(* CODESYS project ugp_spk.project

Project tree, tasks and I/O mapping:
  Device : Owen SPK2xx 03.CS.WEB, Owen, order no. 023, version 3.5.4.20
    application Application
      libraries: Standard, * (System); Util, 3.5.1.0 (System); CmpSysExec, 1.0.0.2 (Owen); ArchiverSPK, 3.5.3.53 (Owen); VisuDialogs, * (System)
      task MainTask (cyclic, interval t#100ms, priority 2) calls PLC_PRG, InterviewState
      task VISU_TASK (cyclic, interval 100 ms, priority 30) calls VisuElems.Visu_Prg
      task AlarmManagerTask (cyclic, interval 50 ms, priority 31) calls AlarmManager.Alarm_Prg
      task bus_task (cyclic, interval t#100ms, priority 1, watchdog t#1000ms x 1) calls MV110
      task LogTask (cyclic, interval t#10000ms, priority 5) calls LogSaver
      program PLC_PRG [ST]
      Alarm Configuration
        alarm class Error (priority 10, acknowledge REP_ACK)
        alarm class Warning (priority 30, acknowledge REP)
        AlarmStorage
        text list AlarmGroup
        alarm group AlarmGroup
            19 [Warning]: Comparison Equal, ExpressionToCompare TRUE, Expression InterviewState.MV110_err - "Нет связи с ЩРПА, ШАСН, ШОПС"
            10 [Warning]: Comparison Equal, ExpressionToCompare TRUE, Expression PLC_PRG.mv110_in_0_alarm_shos - "Нарушение ШОС"
            11 [Warning]: Comparison Equal, ExpressionToCompare TRUE, Expression PLC_PRG.mv110_in_2_alarm_ops - "Авария ОПС"
            12 [Warning]: Comparison Equal, ExpressionToCompare TRUE, Expression PLC_PRG.mpx1_alarm - "Авария ИБПC 2.1"
            13 [Warning]: Comparison Equal, ExpressionToCompare TRUE, Expression PLC_PRG.mpx2_alarm - "Авария ИБПC 2.2"
            14 [Warning]: Comparison Equal, ExpressionToCompare TRUE, Expression PLC_PRG.mv110_in_7_heating - "Обогрев"
            15 [Warning]: Comparison Equal, ExpressionToCompare TRUE, Expression InterviewState.IPS1_err - "Нет связи с ИБПА 1.1"
            16 [Warning]: Comparison Equal, ExpressionToCompare TRUE, Expression InterviewState.IPS2_err - "Нет связи с ИБПА 1.2"
            17 [Warning]: Comparison Equal, ExpressionToCompare TRUE, Expression InterviewState.MPX1_err - "Нет связи с ИБПС 2.1"
            18 [Warning]: Comparison Equal, ExpressionToCompare TRUE, Expression InterviewState.MPX2_err - "Нет связи с ИБПС 2.2"
            9 [Warning]: Comparison Equal, ExpressionToCompare TRUE, Expression PLC_PRG.mv110_in_1_fire - "Пожар"
            20 [Warning]: Comparison Equal, ExpressionToCompare TRUE, Expression PLC_PRG.climate_temp_excess - "Превышена максимальная температура"
      function block Two_words_to_Real [ST]
      visualisation mpx_1_params
      visualisation SCHRPA
      image pool ImagePool
      visualisation mpx_1_state
      visualisation mpx_2_params
      visualisation mpx_2_state
      visualisation main
      visualisation climate
      visualisation SHASN
      visualisation ips_1
      visualisation ips_2
      visualisation alarms
      visualisation log_data
      visualisation SHOPS
      program InterviewState [ST]
      program LogSaver [ST]
    Modbus_COM : Modbus COM, 3S - Smart Software Solutions GmbH, version 3.4.0.0
        settings: DataBits = 8; StopBits = 1; ComPort = 3
      Modbus_Master_COM_Port : Modbus Master, COM Port, 3S - Smart Software Solutions GmbH, version 3.5.5.0
          settings: Transmission = 'RTU'; ResponseTimeout = 1000; TimeBetweenFrames = 10; Auto-restart communication = TRUE
        MV110 : Modbus Slave, COM Port, 3S - Smart Software Solutions GmbH, version 3.5.4.0
            settings: SlaveAddress = 10; ResponseTimeout = 1000; UseExtendedFunctionCodes = TRUE; Channel 0.Function Code = 3; Channel 0.Read Offset = 16#0033; Channel 0.Read Length = 1; Channel 0.Write Offset = 0; Channel 0.Write Length = 0; Channel 0.Cycle Time = 100
            input  Application.PLC_PRG.mv110_reg : WORD  // Channel 0.Channel 0
            unmapped channels: Channel 0
        MPX_1 : Modbus Slave, COM Port, 3S - Smart Software Solutions GmbH, version 3.5.4.0
            settings: SlaveAddress = 11; ResponseTimeout = 1000; UseExtendedFunctionCodes = TRUE; Input_group.Function Code = 4; Input_group.Read Offset = 16#000B; Input_group.Read Length = 7; Input_group.Write Offset = 0; Input_group.Write Length = 0; Input_group.Cycle Time = 300; Bypass_out_group.Function Code = 3; Bypass_out_group.Read Offset = 16#0015; Bypass_out_group.Read Length = 7; Bypass_out_group.Write Offset = 0; Bypass_out_group.Write Length = 0; Bypass_out_group.Cycle Time = 300; Output_group.Function Code = 3; Output_group.Read Offset = 16#001F; Output_group.Read Length = 13; Output_group.Write Offset = 0; Output_group.Write Length = 0; Output_group.Cycle Time = 300; Battery_group.Function Code = 3; Battery_group.Read Offset = 16#002F; Battery_group.Read Length = 7; Battery_group.Write Offset = 0; Battery_group.Write Length = 0; Battery_group.Cycle Time = 300; temp.Function Code = 3; temp.Read Offset = 16#003D; temp.Read Length = 1; temp.Write Offset = 0; temp.Write Length = 0; temp.Cycle Time = 300; states.Function Code = 3; states.Read Offset = 16#0000; states.Read Length = 2; states.Write Offset = 0; states.Write Length = 0; states.Cycle Time = 300; Channel 6.Function Code = 6;
              Channel 6.Read Offset = 0; Channel 6.Read Length = 0; Channel 6.Write Offset = 16#0070; Channel 6.Write Length = 1; Channel 6.Cycle Time = 100
            input  Application.PLC_PRG.mpx1_in_v_1 : WORD  // Input_group.Input_group
            input  Application.PLC_PRG.mpx1_in_v_2 : WORD  // Input_group.Input_group
            input  Application.PLC_PRG.mpx1_in_v_3 : WORD  // Input_group.Input_group
            input  Application.PLC_PRG.mpx1_in_freq : WORD  // Input_group.Input_group
            input  Application.PLC_PRG.mpx1_bypass_v_1 : WORD  // Bypass_out_group.Bypass_out_group
            input  Application.PLC_PRG.mpx1_bypass_v_2 : WORD  // Bypass_out_group.Bypass_out_group
            input  Application.PLC_PRG.mpx1_bypass_v_3 : WORD  // Bypass_out_group.Bypass_out_group
            input  Application.PLC_PRG.mpx1_bypass_freq : WORD  // Bypass_out_group.Bypass_out_group
            input  Application.PLC_PRG.mpx1_output_v_1 : WORD  // Bypass_out_group.Bypass_out_group
            input  Application.PLC_PRG.mpx1_output_v_2 : WORD  // Bypass_out_group.Bypass_out_group
            input  Application.PLC_PRG.mpx1_output_v_3 : WORD  // Bypass_out_group.Bypass_out_group
            input  Application.PLC_PRG.mpx1_output_i_1 : WORD  // Output_group.Output_group
            input  Application.PLC_PRG.mpx1_output_i_2 : WORD  // Output_group.Output_group
            input  Application.PLC_PRG.mpx1_output_i_3 : WORD  // Output_group.Output_group
            input  Application.PLC_PRG.mpx1_load_ph_1 : WORD  // Output_group.Output_group
            input  Application.PLC_PRG.mpx1_load_ph_2 : WORD  // Output_group.Output_group
            input  Application.PLC_PRG.mpx1_load_ph_3 : WORD  // Output_group.Output_group
            input  Application.PLC_PRG.mpx1_output_active_power_1 : WORD  // Output_group.Output_group
            input  Application.PLC_PRG.mpx1_output_active_power_2 : WORD  // Output_group.Output_group
            input  Application.PLC_PRG.mpx1_output_active_power_3 : WORD  // Output_group.Output_group
            input  Application.PLC_PRG.mpx1_output_freq : WORD  // Output_group.Output_group
            input  Application.PLC_PRG.mpx1_battery_voltage : WORD  // Battery_group.Battery_group
            input  Application.PLC_PRG.mpx1_battery_current : WORD  // Battery_group.Battery_group
            input  Application.PLC_PRG.mpx1_battery_capacity : WORD  // Battery_group.Battery_group
            input  Application.PLC_PRG.mpx1_battery_time : WORD  // Battery_group.Battery_group
            input  Application.PLC_PRG.mpx1_temp : WORD  // temp.temp
            input  Application.PLC_PRG.mpx1_state_reg_1 : WORD  // states.states
            input  Application.PLC_PRG.mpx1_state_reg_2 : WORD  // states.states
            output Application.PLC_PRG.mpx_test_battery_start : BIT  // Channel 6
            output Application.PLC_PRG.mpx_test_battery_command : ARRAY[0..0] OF WORD  // Channel 6
            unmapped channels: Input_group, Bypass_out_group, Output_group, Battery_group, temp, states
        MPX_2 : Modbus Slave, COM Port, 3S - Smart Software Solutions GmbH, version 3.5.4.0
            settings: SlaveAddress = 12; ResponseTimeout = 1000; UseExtendedFunctionCodes = TRUE; Input_group.Function Code = 4; Input_group.Read Offset = 16#000B; Input_group.Read Length = 7; Input_group.Write Offset = 0; Input_group.Write Length = 0; Input_group.Cycle Time = 300; Bypass_out_group.Function Code = 3; Bypass_out_group.Read Offset = 16#0015; Bypass_out_group.Read Length = 7; Bypass_out_group.Write Offset = 0; Bypass_out_group.Write Length = 0; Bypass_out_group.Cycle Time = 300; Output_group.Function Code = 3; Output_group.Read Offset = 16#001F; Output_group.Read Length = 13; Output_group.Write Offset = 0; Output_group.Write Length = 0; Output_group.Cycle Time = 300; Battery_group.Function Code = 3; Battery_group.Read Offset = 16#002F; Battery_group.Read Length = 7; Battery_group.Write Offset = 0; Battery_group.Write Length = 0; Battery_group.Cycle Time = 300; temp.Function Code = 3; temp.Read Offset = 16#003D; temp.Read Length = 1; temp.Write Offset = 0; temp.Write Length = 0; temp.Cycle Time = 300; states.Function Code = 3; states.Read Offset = 16#0000; states.Read Length = 2; states.Write Offset = 0; states.Write Length = 0; states.Cycle Time = 300; Channel 6.Function Code = 6;
              Channel 6.Read Offset = 0; Channel 6.Read Length = 0; Channel 6.Write Offset = 16#0070; Channel 6.Write Length = 1; Channel 6.Cycle Time = 100
            input  Application.PLC_PRG.mpx2_in_v_1 : WORD  // Input_group.Input_group
            input  Application.PLC_PRG.mpx2_in_v_2 : WORD  // Input_group.Input_group
            input  Application.PLC_PRG.mpx2_in_v_3 : WORD  // Input_group.Input_group
            input  Application.PLC_PRG.mpx2_in_freq : WORD  // Input_group.Input_group
            input  Application.PLC_PRG.mpx2_bypass_v_1 : WORD  // Bypass_out_group.Bypass_out_group
            input  Application.PLC_PRG.mpx2_bypass_v_2 : WORD  // Bypass_out_group.Bypass_out_group
            input  Application.PLC_PRG.mpx2_bypass_v_3 : WORD  // Bypass_out_group.Bypass_out_group
            input  Application.PLC_PRG.mpx2_bypass_freq : WORD  // Bypass_out_group.Bypass_out_group
            input  Application.PLC_PRG.mpx2_output_v_1 : WORD  // Bypass_out_group.Bypass_out_group
            input  Application.PLC_PRG.mpx2_output_v_2 : WORD  // Bypass_out_group.Bypass_out_group
            input  Application.PLC_PRG.mpx2_output_v_3 : WORD  // Bypass_out_group.Bypass_out_group
            input  Application.PLC_PRG.mpx2_output_i_1 : WORD  // Output_group.Output_group
            input  Application.PLC_PRG.mpx2_output_i_2 : WORD  // Output_group.Output_group
            input  Application.PLC_PRG.mpx2_output_i_3 : WORD  // Output_group.Output_group
            input  Application.PLC_PRG.mpx2_load_ph_1 : WORD  // Output_group.Output_group
            input  Application.PLC_PRG.mpx2_load_ph_2 : WORD  // Output_group.Output_group
            input  Application.PLC_PRG.mpx2_load_ph_3 : WORD  // Output_group.Output_group
            input  Application.PLC_PRG.mpx2_output_active_power_1 : WORD  // Output_group.Output_group
            input  Application.PLC_PRG.mpx2_output_active_power_2 : WORD  // Output_group.Output_group
            input  Application.PLC_PRG.mpx2_output_active_power_3 : WORD  // Output_group.Output_group
            input  Application.PLC_PRG.mpx2_output_freq : WORD  // Output_group.Output_group
            input  Application.PLC_PRG.mpx2_battery_voltage : WORD  // Battery_group.Battery_group
            input  Application.PLC_PRG.mpx2_battery_current : WORD  // Battery_group.Battery_group
            input  Application.PLC_PRG.mpx2_battery_capacity : WORD  // Battery_group.Battery_group
            input  Application.PLC_PRG.mpx2_battery_time : WORD  // Battery_group.Battery_group
            input  Application.PLC_PRG.mpx2_temp : WORD  // temp.temp
            input  Application.PLC_PRG.mpx2_state_reg_1 : WORD  // states.states
            input  Application.PLC_PRG.mpx2_state_reg_2 : WORD  // states.states
            output Application.PLC_PRG.mpx_test_battery_start : BIT  // Channel 6
            output Application.PLC_PRG.mpx_test_battery_command : ARRAY[0..0] OF WORD  // Channel 6
            unmapped channels: Input_group, Bypass_out_group, Output_group, Battery_group, temp, states
    Modbus_slave : Modbus COM, 3S - Smart Software Solutions GmbH, version 3.4.0.0
        settings: DataBits = 8; StopBits = 1; ComPort = 4
      Modbus_Serial_Device : Modbus Serial Device, 3S - Smart Software Solutions GmbH, version 3.5.3.80
          settings: Unit-ID = 3
          output Application.PLC_PRG.mpx1_battery_capacity : WORD  // Outputs.Outputs
          output Application.PLC_PRG.mpx1_battery_current : WORD  // Outputs.Outputs
          output Application.PLC_PRG.mpx1_battery_time : WORD  // Outputs.Outputs
          output Application.PLC_PRG.mpx1_battery_voltage : WORD  // Outputs.Outputs
          output Application.PLC_PRG.mpx1_bypass_freq : WORD  // Outputs.Outputs
          output Application.PLC_PRG.mpx1_bypass_v_1 : WORD  // Outputs.Outputs
          output Application.PLC_PRG.mpx1_bypass_v_2 : WORD  // Outputs.Outputs
          output Application.PLC_PRG.mpx1_bypass_v_3 : WORD  // Outputs.Outputs
          output Application.PLC_PRG.mpx1_in_freq : WORD  // Outputs.Outputs
          output Application.PLC_PRG.mpx1_in_v_1 : WORD  // Outputs.Outputs
          output Application.PLC_PRG.mpx1_in_v_2 : WORD  // Outputs.Outputs
          output Application.PLC_PRG.mpx1_in_v_3 : WORD  // Outputs.Outputs
          output Application.PLC_PRG.mpx1_load_ph_1 : WORD  // Outputs.Outputs
          output Application.PLC_PRG.mpx1_load_ph_2 : WORD  // Outputs.Outputs
          output Application.PLC_PRG.mpx1_load_ph_3 : WORD  // Outputs.Outputs
          output Application.PLC_PRG.mpx1_output_active_power_1 : WORD  // Outputs.Outputs
          output Application.PLC_PRG.mpx1_output_active_power_2 : WORD  // Outputs.Outputs
          output Application.PLC_PRG.mpx1_output_active_power_3 : WORD  // Outputs.Outputs
          output Application.PLC_PRG.mpx1_output_freq : WORD  // Outputs.Outputs
          output Application.PLC_PRG.mpx1_output_i_1 : WORD  // Outputs.Outputs
          output Application.PLC_PRG.mpx1_output_i_2 : WORD  // Outputs.Outputs
          output Application.PLC_PRG.mpx1_output_i_3 : WORD  // Outputs.Outputs
          output Application.PLC_PRG.mpx1_output_v_1 : WORD  // Outputs.Outputs
          output Application.PLC_PRG.mpx1_output_v_2 : WORD  // Outputs.Outputs
          output Application.PLC_PRG.mpx1_output_v_3 : WORD  // Outputs.Outputs
          output Application.PLC_PRG.mpx1_state_reg_1 : WORD  // Outputs.Outputs
          output Application.PLC_PRG.mpx1_state_reg_2 : WORD  // Outputs.Outputs
          output Application.PLC_PRG.mpx1_temp : WORD  // Outputs.Outputs
          output Application.PLC_PRG.mpx2_battery_capacity : WORD  // Outputs.Outputs
          output Application.PLC_PRG.mpx2_battery_current : WORD  // Outputs.Outputs
          output Application.PLC_PRG.mpx2_battery_time : WORD  // Outputs.Outputs
          output Application.PLC_PRG.mpx2_battery_voltage : WORD  // Outputs.Outputs
          output Application.PLC_PRG.mpx2_bypass_freq : WORD  // Outputs.Outputs
          output Application.PLC_PRG.mpx2_bypass_v_1 : WORD  // Outputs.Outputs
          output Application.PLC_PRG.mpx2_bypass_v_2 : WORD  // Outputs.Outputs
          output Application.PLC_PRG.mpx2_bypass_v_3 : WORD  // Outputs.Outputs
          output Application.PLC_PRG.mpx2_in_freq : WORD  // Outputs.Outputs
          output Application.PLC_PRG.mpx2_in_v_1 : WORD  // Outputs.Outputs
          output Application.PLC_PRG.mpx2_in_v_2 : WORD  // Outputs.Outputs
          output Application.PLC_PRG.mpx2_in_v_3 : WORD  // Outputs.Outputs
          output Application.PLC_PRG.mpx2_load_ph_1 : WORD  // Outputs.Outputs
          output Application.PLC_PRG.mpx2_load_ph_2 : WORD  // Outputs.Outputs
          output Application.PLC_PRG.mpx2_load_ph_3 : WORD  // Outputs.Outputs
          output Application.PLC_PRG.mpx2_output_active_power_1 : WORD  // Outputs.Outputs
          output Application.PLC_PRG.mpx2_output_active_power_2 : WORD  // Outputs.Outputs
          output Application.PLC_PRG.mpx2_output_active_power_3 : WORD  // Outputs.Outputs
          output Application.PLC_PRG.mpx2_output_freq : WORD  // Outputs.Outputs
          output Application.PLC_PRG.mpx2_output_i_1 : WORD  // Outputs.Outputs
          output Application.PLC_PRG.mpx2_output_i_2 : WORD  // Outputs.Outputs
          output Application.PLC_PRG.mpx2_output_i_3 : WORD  // Outputs.Outputs
          output Application.PLC_PRG.mpx2_output_v_1 : WORD  // Outputs.Outputs
          output Application.PLC_PRG.mpx2_output_v_2 : WORD  // Outputs.Outputs
          output Application.PLC_PRG.mpx2_output_v_3 : WORD  // Outputs.Outputs
          output Application.PLC_PRG.mpx2_state_reg_1 : WORD  // Outputs.Outputs
          output Application.PLC_PRG.mpx2_state_reg_2 : WORD  // Outputs.Outputs
          output Application.PLC_PRG.mpx2_temp : WORD  // Outputs.Outputs
          output Application.PLC_PRG.ips1_battery_capacity : WORD  // Outputs.Outputs
          output Application.PLC_PRG.ips1_battery_i : WORD  // Outputs.Outputs
          output Application.PLC_PRG.ips1_battery_v : WORD  // Outputs.Outputs
          output Application.PLC_PRG.ips1_bypass_v : WORD  // Outputs.Outputs
          output Application.PLC_PRG.ips1_in_v_1 : WORD  // Outputs.Outputs
          output Application.PLC_PRG.ips1_in_v_2 : WORD  // Outputs.Outputs
          output Application.PLC_PRG.ips1_in_v_3 : WORD  // Outputs.Outputs
          output Application.PLC_PRG.ips1_out_freq : WORD  // Outputs.Outputs
          output Application.PLC_PRG.ips1_out_load : WORD  // Outputs.Outputs
          output Application.PLC_PRG.ips1_out_v : WORD  // Outputs.Outputs
          output Application.PLC_PRG.ips2_battery_capacity : WORD  // Outputs.Outputs
          output Application.PLC_PRG.ips2_battery_i : WORD  // Outputs.Outputs
          output Application.PLC_PRG.ips2_battery_v : WORD  // Outputs.Outputs
          output Application.PLC_PRG.ips2_bypass_v : WORD  // Outputs.Outputs
          output Application.PLC_PRG.ips2_in_v_1 : WORD  // Outputs.Outputs
          output Application.PLC_PRG.ips2_in_v_2 : WORD  // Outputs.Outputs
          output Application.PLC_PRG.ips2_in_v_3 : WORD  // Outputs.Outputs
          output Application.PLC_PRG.ips2_out_freq : WORD  // Outputs.Outputs
          output Application.PLC_PRG.ips2_out_load : WORD  // Outputs.Outputs
          output Application.PLC_PRG.ips2_out_v : WORD  // Outputs.Outputs
          output Application.PLC_PRG.mv110_reg : WORD  // Outputs.Outputs
          output Application.PLC_PRG.climate_state_reg : WORD  // Outputs.Outputs
          output Application.PLC_PRG.climate_temp_in : WORD  // Outputs.Outputs
          output Application.PLC_PRG.climate_temp_out : WORD  // Outputs.Outputs
          unmapped channels: Inputs, Outputs
    Ethernet : Ethernet, 3S - Smart Software Solutions GmbH, version 3.4.2.0
      Modbus_TCP_Master : Modbus TCP Master, 3S - Smart Software Solutions GmbH, version 3.5.4.0
          settings: AutoReconnect = TRUE
        IPS_1 : Modbus TCP Slave, 3S - Smart Software Solutions GmbH, version 3.5.4.0
            settings: Unit-ID = 1; ResponseTimeout = 1500; IPAddress = [192, 168, 19, 34]; Input_group.Function Code = 3; Input_group.Read Offset = 16#006D; Input_group.Read Length = 4; Input_group.Write Offset = 0; Input_group.Write Length = 0; Input_group.Cycle Time = 300; Output_group.Function Code = 3; Output_group.Read Offset = 16#0077; Output_group.Read Length = 5; Output_group.Write Offset = 0; Output_group.Write Length = 0; Output_group.Cycle Time = 300; Bypass_group.Function Code = 3; Bypass_group.Read Offset = 16#0082; Bypass_group.Read Length = 1; Bypass_group.Write Offset = 0; Bypass_group.Write Length = 0; Bypass_group.Cycle Time = 300; Battery_group.Function Code = 3; Battery_group.Read Offset = 16#0063; Battery_group.Read Length = 4; Battery_group.Write Offset = 0; Battery_group.Write Length = 0; Battery_group.Cycle Time = 300
            input  Application.PLC_PRG.ips1_in_v_1 : WORD  // Input_group.Input_group
            input  Application.PLC_PRG.ips1_in_v_2 : WORD  // Input_group.Input_group
            input  Application.PLC_PRG.ips1_in_v_3 : WORD  // Input_group.Input_group
            input  Application.PLC_PRG.ips1_out_freq : WORD  // Output_group.Output_group
            input  Application.PLC_PRG.ips1_out_v : WORD  // Output_group.Output_group
            input  Application.PLC_PRG.ips1_out_load : WORD  // Output_group.Output_group
            input  Application.PLC_PRG.ips1_bypass_v : WORD  // Bypass_group.Bypass_group
            input  Application.PLC_PRG.ips1_battery_v : WORD  // Battery_group.Battery_group
            input  Application.PLC_PRG.ips1_battery_capacity : WORD  // Battery_group.Battery_group
            input  Application.PLC_PRG.ips1_battery_i : WORD  // Battery_group.Battery_group
            unmapped channels: Input_group, Output_group, Bypass_group, Battery_group
        IPS_2 : Modbus TCP Slave, 3S - Smart Software Solutions GmbH, version 3.5.4.0
            settings: Unit-ID = 1; ResponseTimeout = 1500; IPAddress = [192, 168, 19, 35]; Input_group.Function Code = 3; Input_group.Read Offset = 16#006E; Input_group.Read Length = 3; Input_group.Write Offset = 0; Input_group.Write Length = 0; Input_group.Cycle Time = 500; Output_group.Function Code = 3; Output_group.Read Offset = 16#0077; Output_group.Read Length = 7; Output_group.Write Offset = 0; Output_group.Write Length = 0; Output_group.Cycle Time = 500; Bypass_group.Function Code = 3; Bypass_group.Read Offset = 16#0081; Bypass_group.Read Length = 4; Bypass_group.Write Offset = 0; Bypass_group.Write Length = 0; Bypass_group.Cycle Time = 500; Channel 3.Function Code = 3; Channel 3.Read Offset = 16#0063; Channel 3.Read Length = 4; Channel 3.Write Offset = 0; Channel 3.Write Length = 0; Channel 3.Cycle Time = 500
            input  Application.PLC_PRG.ips2_in_v_1 : WORD  // Input_group.Input_group
            input  Application.PLC_PRG.ips2_in_v_2 : WORD  // Input_group.Input_group
            input  Application.PLC_PRG.ips2_in_v_3 : WORD  // Input_group.Input_group
            input  Application.PLC_PRG.ips2_out_freq : WORD  // Output_group.Output_group
            input  Application.PLC_PRG.ips2_out_v : WORD  // Output_group.Output_group
            input  Application.PLC_PRG.ips2_out_load : WORD  // Output_group.Output_group
            input  Application.PLC_PRG.ips2_bypass_v : WORD  // Bypass_group.Bypass_group
            input  Application.PLC_PRG.ips2_battery_v : WORD  // Channel 3.Channel 3
            input  Application.PLC_PRG.ips2_battery_capacity : WORD  // Channel 3.Channel 3
            input  Application.PLC_PRG.ips2_battery_i : WORD  // Channel 3.Channel 3
            unmapped channels: Input_group, Output_group, Bypass_group, Channel 3
    Modbus_PLC_slave : Modbus COM, 3S - Smart Software Solutions GmbH, version 3.4.0.0
        settings: DataBits = 8; StopBits = 1; ComPort = 2
      Modbus_Serial_Device_1 : Modbus Serial Device, 3S - Smart Software Solutions GmbH, version 3.5.5.0
          input  Application.PLC_PRG.climate_temp_in : WORD  // Inputs.Inputs
          input  Application.PLC_PRG.climate_temp_out : WORD  // Inputs.Inputs
          input  Application.PLC_PRG.climate_state_reg : WORD  // Inputs.Inputs
          unmapped channels: Inputs, Outputs
  text list GlobalTextList
  5ce3da45-db07-42e7-a21c-a00fff4ed8f6|C:\workspace\UGP\Images\schrpa.png
  5ce3da45-db07-42e7-a21c-a00fff4ed8f6|D:\scheme_3.png
  5ce3da45-db07-42e7-a21c-a00fff4ed8f6|C:\workspace\UGP\Images\bg_800.png
  5ce3da45-db07-42e7-a21c-a00fff4ed8f6|D:\scheme.png
  5ce3da45-db07-42e7-a21c-a00fff4ed8f6|D:\on.png
  5ce3da45-db07-42e7-a21c-a00fff4ed8f6|D:\off.png
  5ce3da45-db07-42e7-a21c-a00fff4ed8f6|D:\off.jpg
  5ce3da45-db07-42e7-a21c-a00fff4ed8f6|D:\on.jpg
  5ce3da45-db07-42e7-a21c-a00fff4ed8f6|D:\on_ind.jpg
  5ce3da45-db07-42e7-a21c-a00fff4ed8f6|D:\off_ind.jpg
  5ce3da45-db07-42e7-a21c-a00fff4ed8f6|D:\entel.png
  5ce3da45-db07-42e7-a21c-a00fff4ed8f6|D:\zit.png
  5ce3da45-db07-42e7-a21c-a00fff4ed8f6|D:\entel.jpg
  5ce3da45-db07-42e7-a21c-a00fff4ed8f6|D:\zit.jpg
  5ce3da45-db07-42e7-a21c-a00fff4ed8f6|D:\vvod_off.png
  5ce3da45-db07-42e7-a21c-a00fff4ed8f6|D:\vvod_on.png
  5ce3da45-db07-42e7-a21c-a00fff4ed8f6|C:\workspace\UGP\Images\bg.png
  5ce3da45-db07-42e7-a21c-a00fff4ed8f6|C:\workspace\UGP\Images\ups_800.png
  5ce3da45-db07-42e7-a21c-a00fff4ed8f6|C:\workspace\UGP\Images\ups\ups_800.png
  5ce3da45-db07-42e7-a21c-a00fff4ed8f6|C:\workspace\UGP\Images\ups\bypass_line1_off.png
  5ce3da45-db07-42e7-a21c-a00fff4ed8f6|C:\workspace\UGP\Images\ups\bypass_arrow_off.png
  5ce3da45-db07-42e7-a21c-a00fff4ed8f6|C:\workspace\UGP\Images\ups\arrow_off.png
  5ce3da45-db07-42e7-a21c-a00fff4ed8f6|C:\workspace\UGP\Images\ups\battery_arrow_off.png
  5ce3da45-db07-42e7-a21c-a00fff4ed8f6|C:\workspace\UGP\Images\ups\battery_line_off.png
  5ce3da45-db07-42e7-a21c-a00fff4ed8f6|C:\workspace\UGP\Images\ups\battery_arrow_on.png
  5ce3da45-db07-42e7-a21c-a00fff4ed8f6|C:\workspace\UGP\Images\ups\bypass_line_on.png
  5ce3da45-db07-42e7-a21c-a00fff4ed8f6|C:\workspace\UGP\Images\ups\bypass_arrow_on.png
  5ce3da45-db07-42e7-a21c-a00fff4ed8f6|C:\workspace\UGP\Images\ups\arrow_on.png
  5ce3da45-db07-42e7-a21c-a00fff4ed8f6|C:\workspace\UGP\Images\ups\battery_line_on.png
  5ce3da45-db07-42e7-a21c-a00fff4ed8f6|C:\workspace\UGP\Images\main_bg.png
  5ce3da45-db07-42e7-a21c-a00fff4ed8f6|C:\workspace\UGP\Images\shasn.png
  5ce3da45-db07-42e7-a21c-a00fff4ed8f6|C:\workspace\UGP\Images\shasn_1.png
  5ce3da45-db07-42e7-a21c-a00fff4ed8f6|C:\workspace\UGP\Images\ips_state_bg.png
  5ce3da45-db07-42e7-a21c-a00fff4ed8f6|C:\workspace\UGP\Images\mpx_state_bg.png
  5ce3da45-db07-42e7-a21c-a00fff4ed8f6|C:\workspace\UGP\Images\shasn_800.png
*)

// Device/Application/PLC_PRG
PROGRAM PLC_PRG
VAR
	var_test :BOOL:=false;
	alm_1: BOOL;
	alm_2: BOOL;
	war_1: BOOL;
	war_2: BOOL;
	//Переменные для отработки аварийных ситуаций
	accident_sectional_machine :BOOL := FALSE; //авария секционного автомата
	accident_input_1		   :BOOL := FALSE; //авария ввода №1
	accident_input_2		   :BOOL := FALSE; //авария ввода №2
	accident_no_voltage_in_1   :BOOL := FALSE; //отсутствие напряжения на вводе №1
	accident_no_voltage_in_2   :BOOL := FALSE; //отсутствие напряжения на вводе №2
	manual_mode				   :BOOL := FALSE;
	accident_no_voltage_sec    :BOOL := FALSE; //отсутствие напряжения на секции
	
	var_off : BOOL := FALSE;
	var_on : BOOL := TRUE;
	
	//Визуализация
	var_true :BOOL := TRUE;
	ack		 :BOOL;
	history  :BOOL;
	
	//Переменные для работы с MPX_1
	mpx1_in_v_1 	 		   		:WORD; //1-е Напрядение входа
	mpx1_in_v_2 	 		   		:WORD; //2-e Напряжение входа
	mpx1_in_v_3 	 		   		:WORD; //3-е Напряжение входа
	mpx1_in_freq 	 		   		:WORD; //Частота на входе
	mpx1_in_freq_real		   		:REAL; //Частота на входе (x0.1)
	mpx1_bypass_v_1  		   		:WORD; //1-е Напряжение байпаса
	mpx1_bypass_v_2  		   		:WORD; //2-е Напряжение байпаса
	mpx1_bypass_v_3  		   		:WORD; //3-е Напряжение байпаса
	mpx1_bypass_freq 		   		:WORD; //Частота байпаса
	mpx1_bypass_freq_real      		:REAL; //Частота байпаса
	mpx1_output_v_1  		   		:WORD; //1-е Напряжение выхода
	mpx1_output_v_2  		   		:WORD; //2-е Напряжение выхода
	mpx1_output_v_3  		   		:WORD; //3-е Напряжение выхода
	mpx1_output_i_1  		   		:WORD; //1-й Ток выхода
	mpx1_output_i_2  		   		:WORD; //2-й Ток выхода
	mpx1_output_i_3  		   		:WORD; //3-й Ток выхода
	mpx1_output_i_1_real       		:REAL; //1-й Ток выхода (x0.1)
	mpx1_output_i_2_real       		:REAL; //2-й Ток выхода (x0.1)
	mpx1_output_i_3_real       		:REAL; //3-й Ток выхода (x0.1)
	mpx1_output_active_power_1 		:WORD; //Активная мощность 1-й фазы
	mpx1_output_active_power_2 		:WORD; //Активная мощность 2-й фазы
	mpx1_output_active_power_3 		:WORD; //Активная мощность 3-й фазы
	mpx1_output_active_power_1_real :REAL; //Активная мощность 1-й фазы (x0.1)
	mpx1_output_active_power_2_real :REAL; //Активная мощность 2-й фазы (x0.1)
	mpx1_output_active_power_3_real :REAL; //Активная мощность 3-й фазы (x0.1)
	mpx1_output_freq 	       		:WORD; //Частота выхода
	mpx1_output_freq_real 	        :REAL; //Частота выхода (x0.1)
	mpx1_load_ph_1    	       		:WORD; //Загрузска 1-й фазы (%)
	mpx1_load_ph_2    		   		:WORD; //Загрузска 3-й фазы (%)
	mpx1_load_ph_3    	       		:WORD; //Загрузска 2-й фазы (%)
	mpx1_battery_voltage 	   		:WORD; //Напряжение батареи
	mpx1_battery_voltage_real  		:REAL; //Напряжение батареи (x0.1)
	mpx1_battery_current 	   		:WORD; //Ток батареи
	mpx1_battery_current_real  		:REAL; //Ток батареи (x0.1)
	mpx1_battery_capacity 	   		:WORD; //Остаточная емкость батареи (%)
	mpx1_battery_time 		   		:WORD; //Остаточное время автономии (минуты)
	mpx1_temp 				   		:WORD; //Температура
	mpx1_state_reg_1 	       		:WORD; //1-й Регистр состояния
	mpx1_state_1_as_bit 	   		:WORD_AS_BIT;
	mpx1_state_reg_2 		   		:WORD; //2-й Регистр состояния
	mpx1_state_2_as_bit 	   		:WORD_AS_BIT;
	mpx1_bypass_line_state 	   		:STRING; 
	mpx1_bypass_arrow_state    		:STRING;
	mpx1_battery_arrow_state 		:STRING; //состояние батареи
	mpx1_battery_line_state 		:STRING; //состояние батареи
	mpx1_input_state 		   		:STRING; //состояние входа
	mpx1_output_state 		   		:STRING; //состояние выхода
	mpx1_alarm                      :BOOL;
	mpx_test_battery_command        :WORD:=20;
	mpx_test_battery_start          :BOOL;
		
	//Переменные для работы с MPX_2
	mpx2_in_v_1 	 		   		:WORD; //1-е Напрядение входа
	mpx2_in_v_2 	 		   		:WORD; //2-e Напряжение входа
	mpx2_in_v_3 	 		   		:WORD; //3-е Напряжение входа
	mpx2_in_freq 	 		   		:WORD; //Частота на входе
	mpx2_in_freq_real		   		:REAL; //Частота на входе (x0.1)
	mpx2_bypass_v_1  		   		:WORD; //1-е Напряжение байпаса
	mpx2_bypass_v_2  		   		:WORD; //2-е Напряжение байпаса
	mpx2_bypass_v_3  		   		:WORD; //3-е Напряжение байпаса
	mpx2_bypass_freq 		   		:WORD; //Частота байпаса
	mpx2_bypass_freq_real      		:REAL; //Частота байпаса
	mpx2_output_v_1  		   		:WORD; //1-е Напряжение выхода
	mpx2_output_v_2  		   		:WORD; //2-е Напряжение выхода
	mpx2_output_v_3  		   		:WORD; //3-е Напряжение выхода
	mpx2_output_i_1  		   		:WORD; //1-й Ток выхода
	mpx2_output_i_2  		   		:WORD; //2-й Ток выхода
	mpx2_output_i_3  		   		:WORD; //3-й Ток выхода
	mpx2_output_i_1_real       		:REAL; //1-й Ток выхода (x0.1)
	mpx2_output_i_2_real       		:REAL; //2-й Ток выхода (x0.1)
	mpx2_output_i_3_real       		:REAL; //3-й Ток выхода (x0.1)
	mpx2_output_active_power_1 		:WORD; //Активная мощность 1-й фазы
	mpx2_output_active_power_2 		:WORD; //Активная мощность 2-й фазы
	mpx2_output_active_power_3 		:WORD; //Активная мощность 3-й фазы
	mpx2_output_active_power_1_real :REAL; //Активная мощность 1-й фазы (x0.1)
	mpx2_output_active_power_2_real :REAL; //Активная мощность 2-й фазы (x0.1)
	mpx2_output_active_power_3_real :REAL; //Активная мощность 3-й фазы (x0.1)
	mpx2_output_freq 	       		:WORD; //Частота выхода
	mpx2_output_freq_real 	        :REAL; //Частота выхода (x0.1)
	mpx2_load_ph_1    	       		:WORD; //Загрузска 1-й фазы (%)
	mpx2_load_ph_2    		   		:WORD; //Загрузска 3-й фазы (%)
	mpx2_load_ph_3    	       		:WORD; //Загрузска 2-й фазы (%)
	mpx2_battery_voltage 	   		:WORD; //Напряжение батареи
	mpx2_battery_voltage_real  		:REAL; //Напряжение батареи (x0.1)
	mpx2_battery_current 	   		:WORD; //Ток батареи
	mpx2_battery_current_real  		:REAL; //Ток батареи (x0.1)
	mpx2_battery_capacity 	   		:WORD; //Остаточная емкость батареи (%)
	mpx2_battery_time 		   		:WORD; //Остаточное время автономии (минуты)
	mpx2_temp 				   		:WORD; //Температура
	mpx2_state_reg_1 	       		:WORD; //1-й Регистр состояния
	mpx2_state_1_as_bit 	   		:WORD_AS_BIT;
	mpx2_state_reg_2 		   		:WORD; //2-й Регистр состояния
	mpx2_state_2_as_bit 	   		:WORD_AS_BIT;
	mpx2_bypass_line_state 	   		:STRING; 
	mpx2_bypass_arrow_state    		:STRING;
	mpx2_battery_arrow_state 		:STRING; //состояние батареи
	mpx2_battery_line_state 		:STRING; //состояние батареи
	mpx2_input_state 		   		:STRING; //состояние входа
	mpx2_output_state 		   		:STRING; //состояние выхода
	mpx2_alarm                      :BOOL;
	
	//Переменные для работы с климатом
	climate_temp_out        :WORD;
	climat_temp_out_minus   :BOOL; //Регистр отрицательности температуры
	climate_temp_out_real   :REAL;
	climate_temp_in         :WORD;
	climat_temp_in_minus    :BOOL; //Регистр отрицательности температуры
	climate_temp_in_real    :REAL;
	climate_state_reg       :WORD;
	climate_state_as_bit    :WORD_AS_BIT;
	climate_zaslonka_state  :BOOL;
	climate_vent_state      :BOOL;
	climate_condition_state :BOOL;
	climate_heat_state      :BOOL;
	climate_auto_state      :BOOL;
	climate_temp_excess     :BOOL; //авария. внутренняя температура > 25
	
	//Переменные для работы с IPS_1
	ips1_in_v_1           :WORD; //1-е Напряжение входа
	ips1_in_v_1_real      :REAL;
	ips1_in_v_2           :WORD; //2-е Напряжение входа
	ips1_in_v_2_real      :REAL;
	ips1_in_v_3           :WORD; //3-е Напряжение входа
	ips1_in_v_3_real      :REAL;
	ips1_bypass_v         :WORD; //Напряжение байпаса
	ips1_bypass_v_real    :REAL;
	ips1_out_v            :WORD; //Выходное напряжение
	ips1_out_v_real       :REAL;
	ips1_out_freq         :WORD; //Выходная частота
	ips1_out_freq_real    :REAL;
	ips1_out_load         :WORD; //Выходная загрузка
	ips1_out_load_real    :REAL;
	ips1_battery_v        :WORD; //Напряжение батареи
	ips1_battery_v_real   :REAL;
	ips1_battery_capacity :WORD; //Емкость батареи
	ips1_battery_i        :WORD;
	ips1_battery_i_real   :REAL; //Ток батареи
	
	//Переменные для работы с IPS_2
	ips2_in_v_1           :WORD; //1-е Напряжение входа
	ips2_in_v_1_real      :REAL;
	ips2_in_v_2           :WORD; //2-е Напряжение входа
	ips2_in_v_2_real      :REAL;
	ips2_in_v_3           :WORD; //3-е Напряжение входа
	ips2_in_v_3_real      :REAL;
	ips2_bypass_v         :WORD; //Напряжение байпаса
	ips2_bypass_v_real    :REAL;
	ips2_out_v            :WORD; //Выходное напряжение
	ips2_out_v_real       :REAL;
	ips2_out_freq         :WORD; //Выходная частота
	ips2_out_freq_real    :REAL;
	ips2_out_load         :WORD; //Выходная загрузка
	ips2_out_load_real    :REAL;
	ips2_battery_v        :WORD; //Напряжение батареи
	ips2_battery_v_real   :REAL;
	ips2_battery_capacity :WORD; //Емкость батареи
	ips2_battery_i        :WORD;
	ips2_battery_i_real   :REAL; //Ток батареи
	
	//Переменные для работы с первым МВ110-16 (адрес = 1)
	mv110_reg	                   :WORD; //Регистр состояния входов МВ110-16
	mv110_reg_as_bit 	           :WORD_AS_BIT; 
	mv110_in_0_alarm_shos 		   :BOOL; //Нарушение ШОС
	mv110_in_1_fire 			   :BOOL; //Пожар
	mv110_in_2_alarm_ops 		   :BOOL; //Авария ОПС
	mv110_in_3_shasn_main_input    :BOOL; //ШАСН напряжение на основном вводе
	mv110_in_4_shasn_reserve_input :BOOL; //ШАСН напряжение на резервном вводе
	mv110_in_5_shasn_right         :BOOL; //ШАСН напряжение на правой шине
	mv110_in_6_shasn_left          :BOOL; //ШАСН напряжение на левой шине
	mv110_in_7_heating 	           :BOOL; //Обогрев включен
	mv110_in_8_shasn_main 	           :BOOL; //ШАСН основной ввод
	mv110_in_9_shasn_reserve 	           :BOOL; //ШАСН резервный ввод
	mv110_in_10_schrpa_main_input  :BOOL; //ЩРПА напряжение на основном вводе
	mv110_in_11_schrpa_reserve_input  :BOOL; //ЩРПА напряжение на резервном вводе
	mv110_in_12_manual_bypass_1_1   :BOOL; //ЩРПА Ручной байпас 1.1
	mv110_in_12_manual_bypass_1_2  :BOOL; //ЩРПА Ручной байпас 1.2
	
	//Переменные ЩРПА
	schrpa_avr_left_on   :BOOL;
	schrpa_avr_right_on  :BOOL;
	
END_VAR

//Конвертация параметров mpx_1
mpx1_in_freq_real     := mpx1_in_freq * 0.1;
mpx1_bypass_freq_real := mpx1_bypass_freq * 0.1;
mpx1_output_i_1_real  := mpx1_output_i_1 * 0.1;
mpx1_output_i_2_real  := mpx1_output_i_2 * 0.1;
mpx1_output_i_3_real  := mpx1_output_i_3 * 0.1;
mpx1_output_active_power_1_real := mpx1_output_active_power_1 * 0.1;
mpx1_output_active_power_2_real := mpx1_output_active_power_2 * 0.1;
mpx1_output_active_power_3_real := mpx1_output_active_power_3 * 0.1;
mpx1_output_freq_real := mpx1_output_freq * 0.1;
mpx1_battery_voltage_real := mpx1_battery_voltage * 0.1;
mpx1_battery_current_real := mpx1_battery_current * 0.1;

//Логика состояний mpx_1
mpx1_state_1_as_bit(W := mpx1_state_reg_1);
mpx1_state_2_as_bit(W := mpx1_state_reg_2);
IF (mpx1_state_1_as_bit.B11 = FALSE) THEN
	mpx1_bypass_line_state := 'bypass_line1_off';
	mpx1_bypass_arrow_state := 'bypass_arrow_off';
	ELSE
		mpx1_bypass_line_state := 'bypass_line_on';
		mpx1_bypass_arrow_state := 'bypass_arrow_on';	
END_IF
IF (mpx1_state_1_as_bit.B15 = FALSE) THEN
	mpx1_output_state := 'arrow_off';
	ELSE
		mpx1_output_state := 'arrow_on';	
END_IF
IF (mpx1_state_2_as_bit.B12 = FALSE) THEN
	mpx1_input_state := 'arrow_off';
	ELSE
		mpx1_input_state := 'arrow_on';	
END_IF
IF (mpx1_state_1_as_bit.B13 = FALSE) THEN
	mpx1_battery_line_state := 'battery_line_off';
	mpx1_battery_arrow_state := 'battery_arrow_off';
	ELSE
		mpx1_battery_line_state := 'battery_line_on';
		mpx1_battery_arrow_state := 'battery_arrow_on';	
END_IF
IF ( (mpx1_state_2_as_bit.B13 = TRUE) OR (mpx1_state_2_as_bit.B14 = TRUE) OR (mpx1_state_2_as_bit.B15 = TRUE) ) THEN
	mpx1_alarm := TRUE;
	ELSE
		mpx1_alarm := FALSE;
END_IF

//Конвертация параметров mpx_2
mpx2_in_freq_real               := mpx2_in_freq * 0.1;
mpx2_bypass_freq_real           := mpx2_bypass_freq * 0.1;
mpx2_output_i_1_real            := mpx2_output_i_1 * 0.1;
mpx2_output_i_2_real            := mpx2_output_i_2 * 0.1;
mpx2_output_i_3_real            := mpx2_output_i_3 * 0.1;
mpx2_output_active_power_1_real := mpx2_output_active_power_1 * 0.1;
mpx2_output_active_power_2_real := mpx2_output_active_power_2 * 0.1;
mpx2_output_active_power_3_real := mpx2_output_active_power_3 * 0.1;
mpx2_output_freq_real           := mpx2_output_freq * 0.1;
mpx2_battery_voltage_real       := mpx2_battery_voltage * 0.1;
mpx2_battery_current_real       := mpx2_battery_current * 0.1;

//Логика состояний mpx_2
mpx2_state_1_as_bit(W := mpx2_state_reg_1);
mpx2_state_2_as_bit(W := mpx2_state_reg_2);
IF (mpx2_state_1_as_bit.B11 = FALSE) THEN
	mpx2_bypass_line_state := 'bypass_line1_off';
	mpx2_bypass_arrow_state := 'bypass_arrow_off';
	ELSE
		mpx2_bypass_line_state := 'bypass_line_on';
		mpx2_bypass_arrow_state := 'bypass_arrow_on';	
END_IF
IF (mpx2_state_1_as_bit.B15 = FALSE) THEN
	mpx2_output_state := 'arrow_off';
	ELSE
		mpx2_output_state := 'arrow_on';	
END_IF
IF (mpx2_state_2_as_bit.B12 = FALSE) THEN
	mpx2_input_state := 'arrow_off';
	ELSE
		mpx2_input_state := 'arrow_on';	
END_IF
IF (mpx2_state_1_as_bit.B13 = FALSE) THEN
	mpx2_battery_line_state := 'battery_line_off';
	mpx2_battery_arrow_state := 'battery_arrow_off';
	ELSE
		mpx2_battery_line_state := 'battery_line_on';
		mpx2_battery_arrow_state := 'battery_arrow_on';	
END_IF
IF ( (mpx2_state_2_as_bit.B13 = TRUE) OR (mpx2_state_2_as_bit.B14 = TRUE) OR (mpx2_state_2_as_bit.B15 = TRUE) ) THEN
	mpx2_alarm := TRUE;
	ELSE
		mpx2_alarm := FALSE;
END_IF

//Работа с климатом
climate_state_as_bit(W  := climate_state_reg);
climate_zaslonka_state  := climate_state_as_bit.B03;
climate_vent_state      := climate_state_as_bit.B00;
climate_condition_state := climate_state_as_bit.B01;
climate_heat_state      := climate_state_as_bit.B02;
climate_auto_state      := climate_state_as_bit.B04;
climat_temp_out_minus   := climate_state_as_bit.B07;
climat_temp_in_minus    := climate_state_as_bit.B06;
climate_temp_out_real   := climate_temp_out * 0.1;
climate_temp_in_real    := climate_temp_in * 0.1;
IF (climat_temp_out_minus = TRUE) THEN
	climate_temp_out_real := climate_temp_out_real * (-1);
END_IF
IF (climat_temp_in_minus = TRUE) THEN
	climate_temp_in_real := climate_temp_in_real * (-1);
END_IF
IF (climate_temp_in_real > 25) THEN
	climate_temp_excess := TRUE;
	ELSE
		climate_temp_excess := FALSE;
END_IF

//Конвертация ips_1
ips1_in_v_1_real    := ips1_in_v_1 * 0.1;
ips1_in_v_2_real    := ips1_in_v_2 * 0.1;
ips1_in_v_3_real    := ips1_in_v_3 * 0.1;
ips1_bypass_v_real  := ips1_bypass_v * 0.1;
ips1_out_v_real     := ips1_out_v * 0.1;
ips1_out_freq_real  := ips1_out_freq * 0.1;
ips1_battery_v_real := ips1_battery_v * 0.1;
ips1_battery_i_real := ips1_battery_i * 0.1;
ips1_out_load_real  := ips1_out_load * 0.1;

//Конвертация ips_2
ips2_in_v_1_real    := ips2_in_v_1 * 0.1;
ips2_in_v_2_real    := ips2_in_v_2 * 0.1;
ips2_in_v_3_real    := ips2_in_v_3 * 0.1;
ips2_bypass_v_real  := ips2_bypass_v * 0.1;
ips2_out_v_real     := ips2_out_v * 0.1;
ips2_out_freq_real  := ips2_out_freq * 0.1;
ips2_battery_v_real := ips2_battery_v * 0.1;
ips2_battery_i_real := ips2_battery_i * 0.1;
ips2_out_load_real  := ips2_out_load * 0.1;

//Логика МВ110-16
mv110_reg_as_bit(W := mv110_reg);
mv110_in_0_alarm_shos          := mv110_reg_as_bit.B00;
mv110_in_1_fire                := mv110_reg_as_bit.B01;
mv110_in_2_alarm_ops           := mv110_reg_as_bit.B02;
mv110_in_3_shasn_main_input    := mv110_reg_as_bit.B03;
mv110_in_4_shasn_reserve_input := mv110_reg_as_bit.B04;
mv110_in_5_shasn_right         := mv110_reg_as_bit.B05;
mv110_in_6_shasn_left          := mv110_reg_as_bit.B06;
mv110_in_7_heating             := mv110_reg_as_bit.B07;
mv110_in_8_shasn_main             := mv110_reg_as_bit.B08;
mv110_in_9_shasn_reserve             := mv110_reg_as_bit.B09;
mv110_in_10_schrpa_main_input  := mv110_reg_as_bit.B10;
mv110_in_11_schrpa_reserve_input  := mv110_reg_as_bit.B11;
mv110_in_12_manual_bypass_1_1  := mv110_reg_as_bit.B12;
mv110_in_12_manual_bypass_1_2  := mv110_reg_as_bit.B13;

//Логика ЩРПА
IF (mv110_in_10_schrpa_main_input = TRUE) THEN
	schrpa_avr_left_on := TRUE;
	schrpa_avr_right_on := FALSE;
END_IF
IF ( (mv110_in_10_schrpa_main_input = FALSE) AND (mv110_in_11_schrpa_reserve_input = TRUE) ) THEN
	schrpa_avr_left_on := FALSE;
	schrpa_avr_right_on := TRUE;
END_IF
IF ( (mv110_in_10_schrpa_main_input = FALSE) AND (mv110_in_11_schrpa_reserve_input = FALSE) ) THEN
	schrpa_avr_left_on := FALSE;
	schrpa_avr_right_on := FALSE;
END_IF

//Пример конвертации
//module_v1_u1_convertion(Inpit_1:=module_v1_u1_reg1 , Inpit_2:=module_v1_u1_reg2 , output=>module_v1_u1 ); //V1 Ua

END_PROGRAM

// Device/Application/InterviewState
PROGRAM InterviewState
VAR
	MV110_err :BOOL;
	MPX1_err :BOOL;
	MPX2_err :BOOL;
	IPS1_err :BOOL;
	IPS2_err :BOOL;
END_VAR

IF (MV110.xError = TRUE) THEN
	MV110_err := TRUE;
	ELSE
		MV110_err := FALSE;
END_IF

IF (MPX_1.xError = TRUE) THEN
	MPX1_err := TRUE;
	ELSE
		MPX1_err := FALSE;
END_IF

IF (MPX_2.xError = TRUE) THEN
	MPX2_err := TRUE;
	ELSE
		MPX2_err := FALSE;
END_IF

IF (IPS_1.xError = TRUE) THEN
	IPS1_err := TRUE;
	ELSE
		IPS1_err := FALSE;
END_IF

IF (IPS_2.xError = TRUE) THEN
	IPS2_err := TRUE;
	ELSE
		IPS2_err := FALSE;
END_IF

END_PROGRAM

// Device/Application/LogSaver
PROGRAM LogSaver
VAR
	LogArchiver: Archiver;
	ARCH_START :BOOL:=TRUE; //Запуск архивации
	MyDev :StorageDeviseEnum:=Dev_SD1; //Устройства на которое пишется архив
	
	//Архивируемые данные
	ArchiveData: ARRAY[0..63] OF Params_ARCH;

	//Информация
	INFO :WSTRING;
	SDEV_Size :STRING; 
	SDEV_Used :STRING; 
	SDEV_Available :STRING;
END_VAR

//mpx1_in_v_1
ArchiveData[0].dDT :=typeWORD;
ArchiveData[0].pPB :=ADR(PLC_PRG.mpx1_in_v_1);
ArchiveData[0].tTM :=T#180S;

//mpx1_in_v_2
ArchiveData[1].dDT :=typeWORD;
ArchiveData[1].pPB :=ADR(PLC_PRG.mpx1_in_v_2);
ArchiveData[1].tTM :=T#180S;

//mpx1_in_v_3
ArchiveData[2].dDT :=typeWORD;
ArchiveData[2].pPB :=ADR(PLC_PRG.mpx1_in_v_3);
ArchiveData[2].tTM :=T#180S;

//mpx1_bypass_v_1
ArchiveData[3].dDT :=typeWORD;
ArchiveData[3].pPB :=ADR(PLC_PRG.mpx1_bypass_v_1);
ArchiveData[3].tTM :=T#180S;

//mpx1_bypass_v_2
ArchiveData[4].dDT :=typeWORD;
ArchiveData[4].pPB :=ADR(PLC_PRG.mpx1_bypass_v_2);
ArchiveData[4].tTM :=T#180S;

//mpx1_bypass_v_3
ArchiveData[5].dDT :=typeWORD;
ArchiveData[5].pPB :=ADR(PLC_PRG.mpx1_bypass_v_3);
ArchiveData[5].tTM :=T#180S;

//mpx1_output_v_1
ArchiveData[6].dDT :=typeWORD;
ArchiveData[6].pPB :=ADR(PLC_PRG.mpx1_output_v_1);
ArchiveData[6].tTM :=T#180S;

//mpx1_output_v_2
ArchiveData[7].dDT :=typeWORD;
ArchiveData[7].pPB :=ADR(PLC_PRG.mpx1_output_v_2);
ArchiveData[7].tTM :=T#180S;

//mpx1_output_v_3
ArchiveData[8].dDT :=typeWORD;
ArchiveData[8].pPB :=ADR(PLC_PRG.mpx1_output_v_3);
ArchiveData[8].tTM :=T#180S;

//mpx1_output_i_1_real
ArchiveData[9].dDT :=typeREAL;
ArchiveData[9].pPB :=ADR(PLC_PRG.mpx1_output_i_1_real);
ArchiveData[9].tTM :=T#180S;

//mpx1_output_i_2_real
ArchiveData[10].dDT :=typeREAL;
ArchiveData[10].pPB :=ADR(PLC_PRG.mpx1_output_i_2_real);
ArchiveData[10].tTM :=T#180S;

//mpx1_output_i_3_real
ArchiveData[11].dDT :=typeREAL;
ArchiveData[11].pPB :=ADR(PLC_PRG.mpx1_output_i_3_real);
ArchiveData[11].tTM :=T#180S;

//mpx1_output_freq_real
ArchiveData[12].dDT :=typeREAL;
ArchiveData[12].pPB :=ADR(PLC_PRG.mpx1_output_freq_real);
ArchiveData[12].tTM :=T#180S;

//-----------------------------------------------------------------

//mpx2_in_v_1
ArchiveData[13].dDT :=typeWORD;
ArchiveData[13].pPB :=ADR(PLC_PRG.mpx2_in_v_1);
ArchiveData[13].tTM :=T#180S;

//mpx2_in_v_2
ArchiveData[14].dDT :=typeWORD;
ArchiveData[14].pPB :=ADR(PLC_PRG.mpx2_in_v_2);
ArchiveData[14].tTM :=T#180S;

//mpx2_in_v_3
ArchiveData[15].dDT :=typeWORD;
ArchiveData[15].pPB :=ADR(PLC_PRG.mpx2_in_v_3);
ArchiveData[15].tTM :=T#180S;

//mpx2_bypass_v_1
ArchiveData[16].dDT :=typeWORD;
ArchiveData[16].pPB :=ADR(PLC_PRG.mpx2_bypass_v_1);
ArchiveData[16].tTM :=T#180S;

//mpx2_bypass_v_2
ArchiveData[17].dDT :=typeWORD;
ArchiveData[17].pPB :=ADR(PLC_PRG.mpx2_bypass_v_2);
ArchiveData[17].tTM :=T#180S;

//mpx2_bypass_v_3
ArchiveData[18].dDT :=typeWORD;
ArchiveData[18].pPB :=ADR(PLC_PRG.mpx2_bypass_v_3);
ArchiveData[18].tTM :=T#180S;

//mpx2_output_v_1
ArchiveData[19].dDT :=typeWORD;
ArchiveData[19].pPB :=ADR(PLC_PRG.mpx2_output_v_1);
ArchiveData[19].tTM :=T#180S;

//mpx2_output_v_2
ArchiveData[20].dDT :=typeWORD;
ArchiveData[20].pPB :=ADR(PLC_PRG.mpx2_output_v_2);
ArchiveData[20].tTM :=T#180S;

//mpx2_output_v_3
ArchiveData[21].dDT :=typeWORD;
ArchiveData[21].pPB :=ADR(PLC_PRG.mpx2_output_v_3);
ArchiveData[21].tTM :=T#180S;

//mpx2_output_i_1_real
ArchiveData[22].dDT :=typeREAL;
ArchiveData[22].pPB :=ADR(PLC_PRG.mpx2_output_i_1_real);
ArchiveData[22].tTM :=T#180S;

//mpx2_output_i_2_real
ArchiveData[23].dDT :=typeREAL;
ArchiveData[23].pPB :=ADR(PLC_PRG.mpx2_output_i_2_real);
ArchiveData[23].tTM :=T#180S;

//mpx2_output_i_3_real
ArchiveData[24].dDT :=typeREAL;
ArchiveData[24].pPB :=ADR(PLC_PRG.mpx2_output_i_3_real);
ArchiveData[24].tTM :=T#180S;

//mpx2_output_freq_real
ArchiveData[25].dDT :=typeREAL;
ArchiveData[25].pPB :=ADR(PLC_PRG.mpx2_output_freq_real);
ArchiveData[25].tTM :=T#180S;

//-----------------------------------------------------------------

//ips1_in_v_1_real
ArchiveData[26].dDT :=typeREAL;
ArchiveData[26].pPB :=ADR(PLC_PRG.ips1_in_v_1_real);
ArchiveData[26].tTM :=T#180S;

//ips1_in_v_2_real
ArchiveData[27].dDT :=typeREAL;
ArchiveData[27].pPB :=ADR(PLC_PRG.ips1_in_v_2_real);
ArchiveData[27].tTM :=T#180S;

//ips1_in_v_3_real
ArchiveData[28].dDT :=typeREAL;
ArchiveData[28].pPB :=ADR(PLC_PRG.ips1_in_v_3_real);
ArchiveData[28].tTM :=T#180S;

//ips1_bypass_v_real
ArchiveData[29].dDT :=typeREAL;
ArchiveData[29].pPB :=ADR(PLC_PRG.ips1_bypass_v_real);
ArchiveData[29].tTM :=T#180S;

//ips1_out_v_real
ArchiveData[30].dDT :=typeREAL;
ArchiveData[30].pPB :=ADR(PLC_PRG.ips1_out_v_real);
ArchiveData[30].tTM :=T#180S;

//ips1_out_freq_real
ArchiveData[31].dDT :=typeREAL;
ArchiveData[31].pPB :=ADR(PLC_PRG.ips1_out_freq_real);
ArchiveData[31].tTM :=T#180S;

//ips1_out_load_real
ArchiveData[32].dDT :=typeREAL;
ArchiveData[32].pPB :=ADR(PLC_PRG.ips1_out_load_real);
ArchiveData[32].tTM :=T#180S;

//-----------------------------------------------------------------

//ips2_in_v_1_real
ArchiveData[33].dDT :=typeREAL;
ArchiveData[33].pPB :=ADR(PLC_PRG.ips2_in_v_1_real);
ArchiveData[33].tTM :=T#180S;

//ips2_in_v_2_real
ArchiveData[34].dDT :=typeREAL;
ArchiveData[34].pPB :=ADR(PLC_PRG.ips2_in_v_2_real);
ArchiveData[34].tTM :=T#180S;

//ips2_in_v_3_real
ArchiveData[35].dDT :=typeREAL;
ArchiveData[35].pPB :=ADR(PLC_PRG.ips2_in_v_3_real);
ArchiveData[35].tTM :=T#180S;

//ips2_bypass_v_real
ArchiveData[36].dDT :=typeREAL;
ArchiveData[36].pPB :=ADR(PLC_PRG.ips2_bypass_v_real);
ArchiveData[36].tTM :=T#180S;

//ips2_out_v_real
ArchiveData[37].dDT :=typeREAL;
ArchiveData[37].pPB :=ADR(PLC_PRG.ips2_out_v_real);
ArchiveData[37].tTM :=T#180S;

//ips2_out_freq_real
ArchiveData[38].dDT :=typeREAL;
ArchiveData[38].pPB :=ADR(PLC_PRG.ips2_out_freq_real);
ArchiveData[38].tTM :=T#180S;

//ips2_out_load_real
ArchiveData[39].dDT :=typeREAL;
ArchiveData[39].pPB :=ADR(PLC_PRG.ips2_out_load_real);
ArchiveData[39].tTM :=T#180S;

//-----------------------------------------------------------------

//climate_temp_out_real
ArchiveData[40].dDT :=typeREAL;
ArchiveData[40].pPB :=ADR(PLC_PRG.climate_temp_out_real);
ArchiveData[40].tTM :=T#180S;

//climate_temp_in_real
ArchiveData[41].dDT :=typeREAL;
ArchiveData[41].pPB :=ADR(PLC_PRG.climate_temp_in_real);
ArchiveData[41].tTM :=T#180S;

LogArchiver(
	Start:= ARCH_START, 
	TypeDevice:= MyDev, 
	ARCH_Data:= ArchiveData, 
	TypeDeviceForCopy:= , 
	Copy:= , 
	INFO=> INFO, 
	DEV_Size=> , 
	DEV_Used=> , 
	DEV_Available=> , 
	DEV_Use=> , 
	SDEV_Size=> SDEV_Size, 
	SDEV_Used=> SDEV_Used, 
	SDEV_Available=> SDEV_Available, 
	All_Err=> , 
	DevStatus=> , 
	Done=> );

END_PROGRAM

// Device/Application/Two_words_to_Real
FUNCTION_BLOCK Two_words_to_Real
VAR_INPUT
	Inpit_1:WORD;
	Inpit_2:WORD;
END_VAR
VAR_OUTPUT
	output:real;
END_VAR
VAR
	P:POINTER TO ARRAY [0..3] OF BYTE; 
	pi1:POINTER TO ARRAY [0..1] OF BYTE; 
	pi2:POINTER TO ARRAY [0..1] OF BYTE; 
END_VAR

pi1:=ADR(Inpit_1);
pi2:=ADR(Inpit_2);



P:=ADR(output);
P^[0]:=pi2^[0];
P^[1]:=pi2^[1];
P^[2]:=pi1^[0];
P^[3]:=pi1^[1];

END_FUNCTION_BLOCK

// Device/Application/mpx_1_params
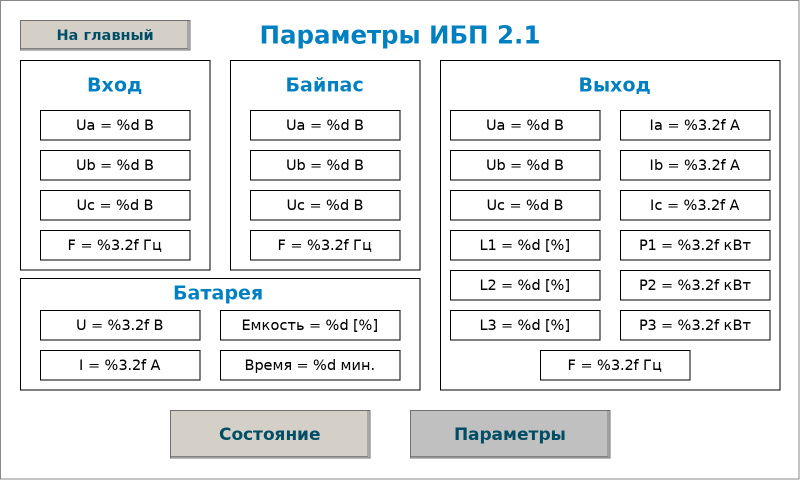
VISUALIZATION mpx_1_params  // 800x480, background image ImagePool.bg_800
    Rectangle (186,20 428x30), "Параметры ИБП 2.1"
    Button (170,410 200x48), "Состояние"
        OnMouseClick:  Assign=mpx_1_state, Type=Assignment
    Button (410,410 200x48), "Параметры", pressed state: PLC_PRG.var_true
    Button (20,20 170x30), "На главный"
        OnMouseClick:  Assign=main, Type=Assignment
    Rectangle (20,60 190x210)
    Rectangle (440,60 340x330)
    Rectangle (30,70 170x30), "Вход"
    Rectangle (40,110 150x30), "Ua = %d В", text variable: PLC_PRG.mpx1_in_v_1
    Rectangle (40,150 150x30), "Ub = %d В", text variable: PLC_PRG.mpx1_in_v_2
    Rectangle (40,190 150x30), "Uc = %d В", text variable: PLC_PRG.mpx1_in_v_3
    Rectangle (40,230 150x30), "F = %3.2f Гц", text variable: PLC_PRG.mpx1_in_freq_real
    Rectangle (230,60 190x210)
    Rectangle (240,70 170x30), "Байпас"
    Rectangle (250,110 150x30), "Ua = %d В", text variable: PLC_PRG.mpx1_bypass_v_1
    Rectangle (250,150 150x30), "Ub = %d В", text variable: PLC_PRG.mpx1_bypass_v_2
    Rectangle (250,190 150x30), "Uc = %d В", text variable: PLC_PRG.mpx1_bypass_v_3
    Rectangle (250,230 150x30), "F = %3.2f Гц", text variable: PLC_PRG.mpx1_bypass_freq_real
    Rectangle (460,70 310x30), "Выход"
    Rectangle (450,110 150x30), "Ua = %d В", text variable: PLC_PRG.mpx1_output_v_1
    Rectangle (450,150 150x30), "Ub = %d В", text variable: PLC_PRG.mpx1_output_v_2
    Rectangle (450,190 150x30), "Uc = %d В", text variable: PLC_PRG.mpx1_output_v_3
    Rectangle (620,110 150x30), "Ia = %3.2f A", text variable: PLC_PRG.mpx1_output_i_1_real
    Rectangle (620,150 150x30), "Ib = %3.2f A", text variable: PLC_PRG.mpx1_output_i_2_real
    Rectangle (620,190 150x30), "Ic = %3.2f A", text variable: PLC_PRG.mpx1_output_i_3_real
    Rectangle (450,230 150x30), "L1 = %d [%]", text variable: PLC_PRG.mpx1_load_ph_1
    Rectangle (450,270 150x30), "L2 = %d [%]", text variable: PLC_PRG.mpx1_load_ph_2
    Rectangle (450,310 150x30), "L3 = %d [%]", text variable: PLC_PRG.mpx1_load_ph_3
    Rectangle (620,230 150x30), "P1 = %3.2f кВт", text variable: PLC_PRG.mpx1_output_active_power_1_real
    Rectangle (620,270 150x30), "P2 = %3.2f кВт", text variable: PLC_PRG.mpx1_output_active_power_2_real
    Rectangle (620,310 150x30), "P3 = %3.2f кВт", text variable: PLC_PRG.mpx1_output_active_power_3_real
    Rectangle (540,350 150x30), "F = %3.2f Гц", text variable: PLC_PRG.mpx1_output_freq_real
    Rectangle (20,278 400x112)
    Rectangle (30,284 376x18), "Батарея"
    Rectangle (40,310 160x30), "U = %3.2f В", text variable: PLC_PRG.mpx1_battery_voltage_real
    Rectangle (40,350 160x30), "I = %3.2f A", text variable: PLC_PRG.mpx1_battery_current_real
    Rectangle (220,310 180x30), "Емкость = %d [%]", text variable: PLC_PRG.mpx1_battery_capacity
    Rectangle (220,350 180x30), "Время = %d мин.", text variable: PLC_PRG.mpx1_battery_time
    hotkey  Id=481037385728, Key=KeyDown=True, KeyName=0
    hotkey  Id=481038434304, Key=KeyName=0
END_VISUALIZATION

// Device/Application/SCHRPA
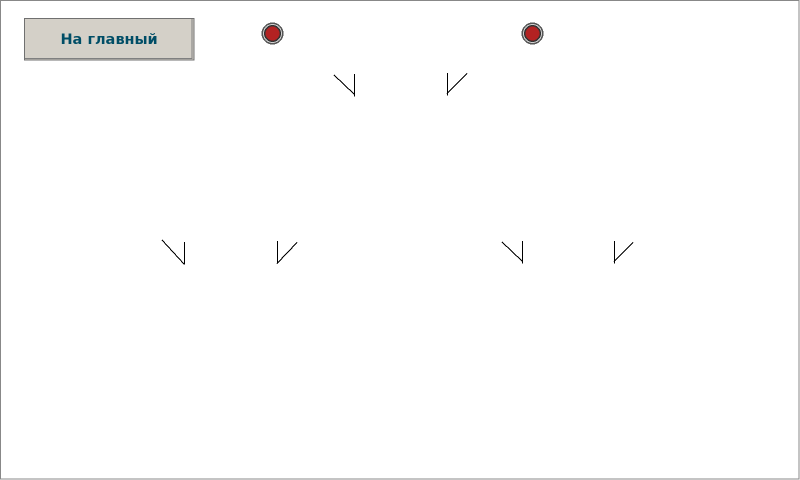
VISUALIZATION SCHRPA  // 800x480, background image ImagePool.schrpa_bg
    Button (24,18 170x42), "На главный"
        OnMouseClick:  Assign=main, Type=Assignment
    Line (150,240)
    Line (184,264) (162,240), invisible if: NOT(PLC_PRG.mv110_in_12_manual_bypass_1_1)
    Line (184,242) (184,264), invisible if: PLC_PRG.mv110_in_12_manual_bypass_1_1
    Line (277,263) (297,242), invisible if: PLC_PRG.mv110_in_12_manual_bypass_1_1
    Line (277,241) (277,263), invisible if: NOT(PLC_PRG.mv110_in_12_manual_bypass_1_1)
    Line (354,74) (354,96), invisible if: NOT(PLC_PRG.schrpa_avr_left_on)
    Line (447,73) (447,95), invisible if: NOT(PLC_PRG.schrpa_avr_right_on)
    Line (354,94) (334,75), invisible if: PLC_PRG.schrpa_avr_left_on
    Line (447,93) (467,73), invisible if: PLC_PRG.schrpa_avr_right_on
    Line (522,241) (522,263), invisible if: NOT(PLC_PRG.mv110_in_12_manual_bypass_1_2)
    Line (522,261) (502,242), invisible if: PLC_PRG.mv110_in_12_manual_bypass_1_2
    Line (614,241) (614,263), invisible if: PLC_PRG.mv110_in_12_manual_bypass_1_2
    Line (614,261) (633,242), invisible if: NOT(PLC_PRG.mv110_in_12_manual_bypass_1_2)
    Lamp1 (260,20 25x27), variable: PLC_PRG.mv110_in_10_schrpa_main_input, style: Lamp-Lamp1-Red
    Lamp1 (520,20 25x27), variable: PLC_PRG.mv110_in_11_schrpa_reserve_input, style: Lamp-Lamp1-Red
    hotkey  Id=481037385728, Key=KeyDown=True, KeyName=0, VisuElemId=1
    hotkey  Id=481038434304, Key=KeyName=0, VisuElemId=1
END_VISUALIZATION

// Device/Application/mpx_1_state
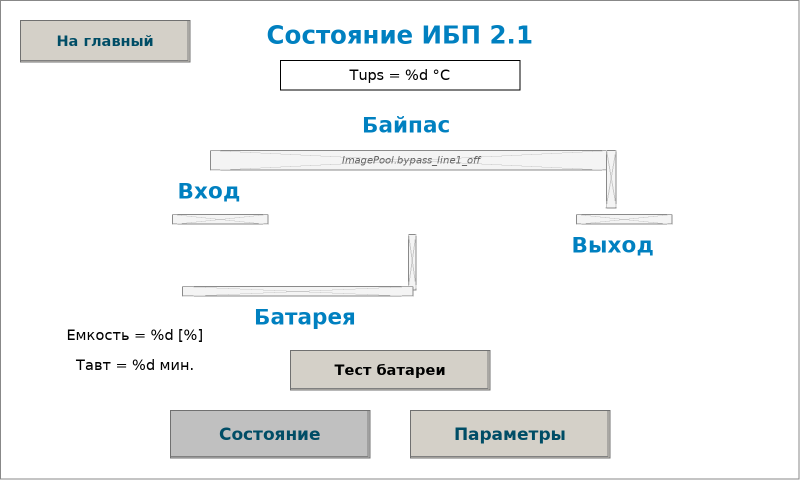
VISUALIZATION mpx_1_state  // 800x480, background image ImagePool.mpx_state_bg
    Rectangle (186,20 428x30), "Состояние ИБП 2.1"
    Button (410,410 200x48), "Параметры"
        OnMouseClick:  Assign=mpx_1_params, Type=Assignment
    Button (170,410 200x48), "Состояние", pressed state: PLC_PRG.var_true
    Button (20,20 170x42), "На главный"
        OnMouseClick:  Assign=main, Type=Assignment
    Rectangle (350,110 112x30), "Байпас"
    Rectangle (246,302 118x30), "Батарея"
    Rectangle (166,176 86x30), "Вход"
    Rectangle (560,230 106x30), "Выход"
    Rectangle (280,60 240x30), "Tups = %d °С", text variable: PLC_PRG.mpx1_temp
    Rectangle (30,320 210x30), "Емкость = %d [%]", text variable: PLC_PRG.mpx1_battery_capacity
    Rectangle (30,350 210x30), "Tавт = %d мин.", text variable: PLC_PRG.mpx1_battery_time
    Image (210,150 402x20), image: ImagePool.bypass_line1_off
        p84334746: PLC_PRG.mpx1_bypass_line_state
    Image (606,150 10x58), image: ImagePool.bypass_arrow_off
        p84334746: PLC_PRG.mpx1_bypass_arrow_state
    Image (576,214 96x10), image: ImagePool.arrow_off
        p84334746: PLC_PRG.mpx1_output_state
    Image (172,214 96x10), image: ImagePool.arrow_off
        p84334746: PLC_PRG.mpx1_input_state
    Image (408,234 8x56), image: ImagePool.battery_arrow_off
        p84334746: PLC_PRG.mpx1_battery_arrow_state
    Image (182,286 231x10), image: ImagePool.battery_line_off
        p84334746: PLC_PRG.mpx1_battery_line_state
    Button (290,350 200x40), "Тест батареи"
        OnMouseClick:  ToggleVariable=PLC_PRG.mpx_test_battery_start
    hotkey  Id=481037385728, Key=KeyDown=True, KeyName=0, VisuElemId=91
    hotkey  Id=481038434304, Key=KeyName=0, VisuElemId=91
END_VISUALIZATION

// Device/Application/mpx_2_params
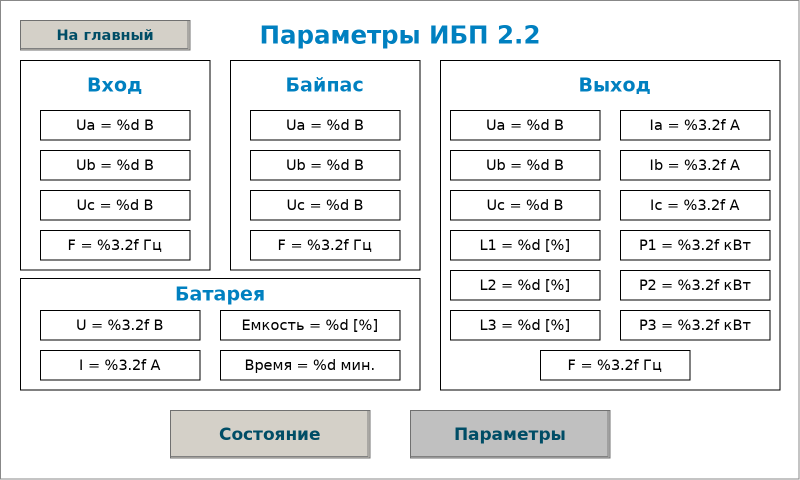
VISUALIZATION mpx_2_params  // 800x480, background image ImagePool.bg_800
    Rectangle (186,20 428x30), "Параметры ИБП 2.2"
    Button (170,410 200x48), "Состояние"
        OnMouseClick:  Assign=mpx_2_state, Type=Assignment
    Button (410,410 200x48), "Параметры", pressed state: PLC_PRG.var_true
    Button (20,20 170x30), "На главный"
        OnMouseClick:  Assign=main, Type=Assignment
    Rectangle (20,60 190x210)
    Rectangle (440,60 340x330)
    Rectangle (30,70 170x30), "Вход"
    Rectangle (40,110 150x30), "Ua = %d В", text variable: PLC_PRG.mpx2_in_v_1
    Rectangle (40,150 150x30), "Ub = %d В", text variable: PLC_PRG.mpx2_in_v_2
    Rectangle (40,190 150x30), "Uc = %d В", text variable: PLC_PRG.mpx2_in_v_3
    Rectangle (40,230 150x30), "F = %3.2f Гц", text variable: PLC_PRG.mpx2_in_freq_real
    Rectangle (230,60 190x210)
    Rectangle (240,70 170x30), "Байпас"
    Rectangle (250,110 150x30), "Ua = %d В", text variable: PLC_PRG.mpx2_bypass_v_1
    Rectangle (250,150 150x30), "Ub = %d В", text variable: PLC_PRG.mpx2_bypass_v_2
    Rectangle (250,190 150x30), "Uc = %d В", text variable: PLC_PRG.mpx2_bypass_v_3
    Rectangle (250,230 150x30), "F = %3.2f Гц", text variable: PLC_PRG.mpx2_bypass_freq_real
    Rectangle (460,70 310x30), "Выход"
    Rectangle (450,110 150x30), "Ua = %d В", text variable: PLC_PRG.mpx2_output_v_1
    Rectangle (450,150 150x30), "Ub = %d В", text variable: PLC_PRG.mpx2_output_v_2
    Rectangle (450,190 150x30), "Uc = %d В", text variable: PLC_PRG.mpx2_output_v_3
    Rectangle (620,110 150x30), "Ia = %3.2f A", text variable: PLC_PRG.mpx2_output_i_1_real
    Rectangle (620,150 150x30), "Ib = %3.2f A", text variable: PLC_PRG.mpx2_output_i_2_real
    Rectangle (620,190 150x30), "Ic = %3.2f A", text variable: PLC_PRG.mpx2_output_i_3_real
    Rectangle (450,230 150x30), "L1 = %d [%]", text variable: PLC_PRG.mpx2_load_ph_1
    Rectangle (450,270 150x30), "L2 = %d [%]", text variable: PLC_PRG.mpx2_load_ph_2
    Rectangle (450,310 150x30), "L3 = %d [%]", text variable: PLC_PRG.mpx2_load_ph_3
    Rectangle (620,230 150x30), "P1 = %3.2f кВт", text variable: PLC_PRG.mpx2_output_active_power_1_real
    Rectangle (620,270 150x30), "P2 = %3.2f кВт", text variable: PLC_PRG.mpx2_output_active_power_2_real
    Rectangle (620,310 150x30), "P3 = %3.2f кВт", text variable: PLC_PRG.mpx2_output_active_power_3_real
    Rectangle (540,350 150x30), "F = %3.2f Гц", text variable: PLC_PRG.mpx2_output_freq_real
    Rectangle (20,278 400x112)
    Rectangle (30,282 380x24), "Батарея"
    Rectangle (40,310 160x30), "U = %3.2f В", text variable: PLC_PRG.mpx2_battery_voltage_real
    Rectangle (40,350 160x30), "I = %3.2f A", text variable: PLC_PRG.mpx2_battery_current_real
    Rectangle (220,310 180x30), "Емкость = %d [%]", text variable: PLC_PRG.mpx2_battery_capacity
    Rectangle (220,350 180x30), "Время = %d мин.", text variable: PLC_PRG.mpx2_battery_time
    hotkey  Id=481037385728, Key=KeyDown=True, KeyName=0
    hotkey  Id=481038434304, Key=KeyName=0
END_VISUALIZATION

// Device/Application/mpx_2_state
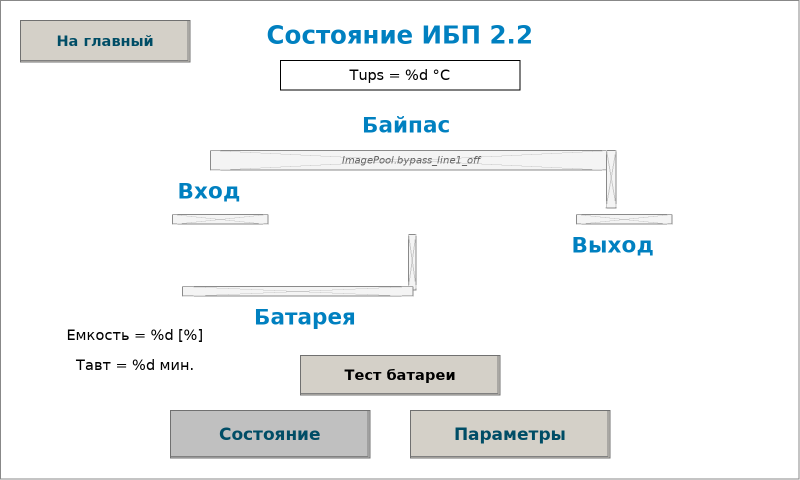
VISUALIZATION mpx_2_state  // 800x480, background image ImagePool.mpx_state_bg
    Rectangle (186,20 428x30), "Состояние ИБП 2.2"
    Button (410,410 200x48), "Параметры"
        OnMouseClick:  Assign=mpx_2_params, Type=Assignment
    Button (170,410 200x48), "Состояние", pressed state: PLC_PRG.var_true
    Button (20,20 170x42), "На главный"
        OnMouseClick:  Assign=main, Type=Assignment
    Rectangle (350,110 112x30), "Байпас"
    Rectangle (246,302 118x30), "Батарея"
    Rectangle (166,176 86x30), "Вход"
    Rectangle (560,230 106x30), "Выход"
    Rectangle (280,60 240x30), "Tups = %d °С", text variable: PLC_PRG.mpx2_temp
    Rectangle (30,320 210x30), "Емкость = %d [%]", text variable: PLC_PRG.mpx2_battery_capacity
    Rectangle (30,350 210x30), "Tавт = %d мин.", text variable: PLC_PRG.mpx2_battery_time
    Image (210,150 402x20), image: ImagePool.bypass_line1_off
        p84334746: PLC_PRG.mpx2_bypass_line_state
    Image (606,150 10x58), image: ImagePool.bypass_arrow_off
        p84334746: PLC_PRG.mpx2_bypass_arrow_state
    Image (576,214 96x10), image: ImagePool.arrow_off
        p84334746: PLC_PRG.mpx2_output_state
    Image (172,214 96x10), image: ImagePool.arrow_off
        p84334746: PLC_PRG.mpx2_input_state
    Image (408,234 8x56), image: ImagePool.battery_arrow_off
        p84334746: PLC_PRG.mpx2_battery_arrow_state
    Image (182,286 231x10), image: ImagePool.battery_line_off
        p84334746: PLC_PRG.mpx2_battery_line_state
    Button (300,355 200x40), "Тест батареи"
        OnMouseClick:  ToggleVariable=PLC_PRG.mpx_test_battery_start
    hotkey  Id=481037385728, Key=KeyDown=True, KeyName=0, VisuElemId=91
    hotkey  Id=481038434304, Key=KeyName=0, VisuElemId=91
END_VISUALIZATION

// Device/Application/main
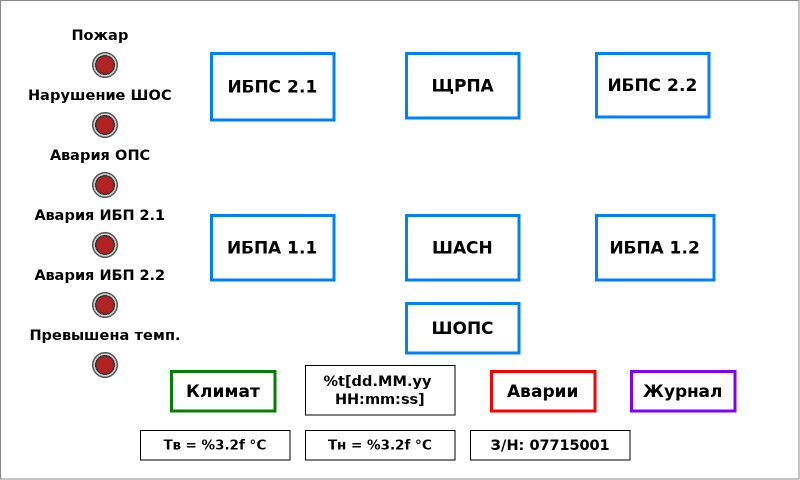
VISUALIZATION main  // 800x480, background image ImagePool.main_bg
    RoundedRectangle (210,52 125x69), "ИБПС 2.1", colour toggle: InterviewState.MPX1_err
        OnMouseClick:  Assign=mpx_1_state, Type=Assignment
    RoundedRectangle (595,52 115x66), "ИБПС 2.2", colour toggle: InterviewState.MPX2_err
        OnMouseClick:  Assign=mpx_2_state, Type=Assignment
    RoundedRectangle (170,370 106x42), "Климат"
        OnMouseClick:  Assign=climate, Type=Assignment
    RoundedRectangle (405,214 115x67), "ШАСН", colour toggle: InterviewState.MV110_err
        OnMouseClick:  Assign=SHASN, Type=Assignment
    RoundedRectangle (210,214 125x67), "ИБПА 1.1", colour toggle: InterviewState.IPS1_err
        OnMouseClick:  Assign=ips_1, Type=Assignment
    RoundedRectangle (595,214 120x67), "ИБПА 1.2", colour toggle: InterviewState.IPS2_err
        OnMouseClick:  Assign=ips_2, Type=Assignment
    RoundedRectangle (405,52 115x67), "ЩРПА", colour toggle: InterviewState.MV110_err
        OnMouseClick:  Assign=SCHRPA, Type=Assignment
    RoundedRectangle (490,370 106x42), "Аварии"
        OnMouseClick:  Assign=alarms, Type=Assignment
    Lamp1 (90,50 30x30), variable: PLC_PRG.mv110_in_1_fire, style: Lamp-Lamp1-Red
    Rectangle (20,20 160x30), "Пожар"
    Lamp1 (90,110 30x30), variable: PLC_PRG.mv110_in_0_alarm_shos, style: Lamp-Lamp1-Red
    Rectangle (20,80 160x30), "Нарушение ШОС"
    Lamp1 (90,170 30x30), variable: PLC_PRG.mv110_in_2_alarm_ops, style: Lamp-Lamp1-Red
    Rectangle (20,140 160x30), "Авария ОПС"
    Lamp1 (90,230 30x30), variable: PLC_PRG.mpx1_alarm, style: Lamp-Lamp1-Red
    Rectangle (20,200 160x30), "Авария ИБП 2.1"
    Lamp1 (90,290 30x30), variable: PLC_PRG.mpx2_alarm, style: Lamp-Lamp1-Red
    Rectangle (20,260 160x30), "Авария ИБП 2.2"
    RoundedRectangle (405,302 115x52), "ШОПС", colour toggle: InterviewState.MV110_err
        OnMouseClick:  Assign=SHOPS, Type=Assignment
    Lamp1 (90,350 30x30), variable: PLC_PRG.climate_temp_excess, style: Lamp-Lamp1-Red
    Rectangle (20,320 170x30), "Превышена темп."
    Rectangle (470,430 160x30), "З/Н: 07715001"
    Rectangle (140,430 150x30), "Tв = %3.2f °С", text variable: PLC_PRG.climate_temp_in_real
    Rectangle (305,430 150x30), "Tн = %3.2f °С", text variable: PLC_PRG.climate_temp_out_real
    Rectangle (305,365 150x50), "%t[dd.MM.yy HH:mm:ss]"
    RoundedRectangle (630,370 106x42), "Журнал"
        OnMouseClick:  Assign=log_data, Type=Assignment
END_VISUALIZATION

// Device/Application/climate
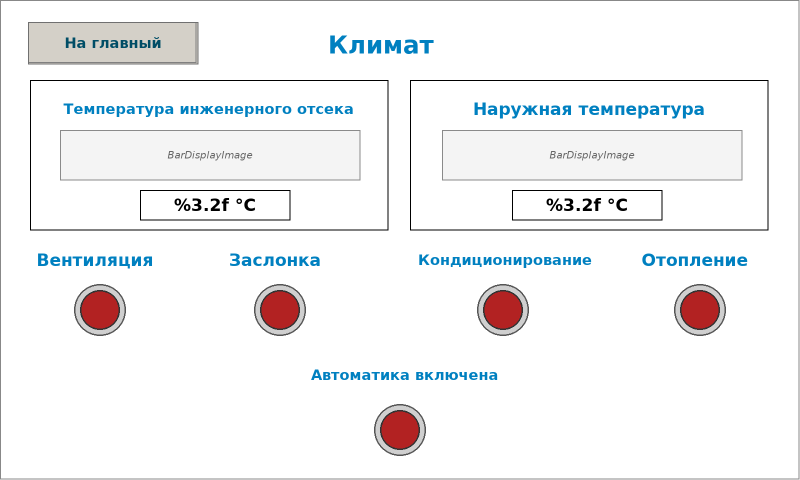
VISUALIZATION climate  // 800x480, background image ImagePool.bg_800
    Rectangle (220,30 322x30), "Климат"
    Button (28,22 170x42), "На главный"
        OnMouseClick:  Assign=main, Type=Assignment
    Rectangle (30,80 358x150), text variable: PLC_PRG.mpx1_bypass_v_1
    Rectangle (36,94 346x30), "Температура инженерного отсека"
    Rectangle (140,190 150x30), "%3.2f °С", text variable: PLC_PRG.climate_temp_in_real
    BarDisplayImage (60,130 300x50), value: PLC_PRG.climate_temp_in_real, style: BarDisplayImage-Gray, scale format: %.1f, scale -10..50
    Rectangle (410,80 358x150), text variable: PLC_PRG.mpx1_bypass_v_1
    Rectangle (416,94 346x30), "Наружная температура"
    Rectangle (512,190 150x30), "%3.2f °С", text variable: PLC_PRG.climate_temp_out_real
    BarDisplayImage (442,130 300x50), value: PLC_PRG.climate_temp_out_real, style: BarDisplayImage-Gray, scale format: %.1f, scale -60..80
    Rectangle (270,360 270x30), "Автоматика включена"
    Lamp1 (370,400 60x60), variable: PLC_PRG.climate_auto_state, style: Lamp-Lamp1-Red
    Lamp1 (70,280 60x60), variable: PLC_PRG.climate_vent_state, style: Lamp-Lamp1-Red
    Rectangle (20,250 150x20), "Вентиляция"
    Lamp1 (250,280 60x60), variable: PLC_PRG.climate_zaslonka_state, style: Lamp-Lamp1-Red
    Rectangle (220,250 110x20), "Заслонка"
    Rectangle (400,250 210x20), "Кондиционирование"
    Lamp1 (470,280 66x60), variable: PLC_PRG.climate_condition_state, style: Lamp-Lamp1-Red
    Lamp1 (670,280 60x60), variable: PLC_PRG.climate_heat_state, style: Lamp-Lamp1-Red
    Rectangle (620,250 150x20), "Отопление"
    hotkey  Id=481037385728, Key=KeyDown=True, KeyName=0, VisuElemId=3
    hotkey  Id=481038434304, Key=KeyName=0, VisuElemId=3
END_VISUALIZATION

// Device/Application/SHASN
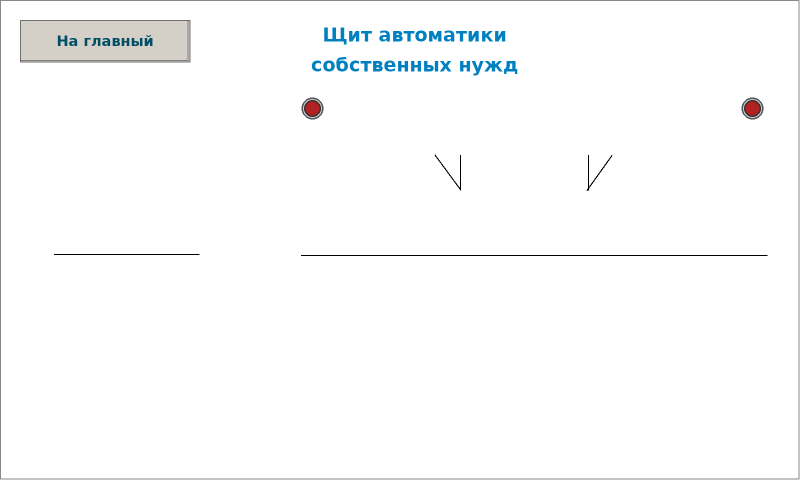
VISUALIZATION SHASN  // 800x480, background image ImagePool.shasn_bg
    Rectangle (260,20 310x30), "Щит автоматики"
    Rectangle (260,50 310x30), "собственных нужд"
    Button (20,20 170x42), "На главный"
        OnMouseClick:  Assign=main, Type=Assignment
    Lamp1 (300,95 25x27), variable: PLC_PRG.mv110_in_3_shasn_main_input, style: Lamp-Lamp1-Red
    Lamp1 (740,95 25x27), variable: PLC_PRG.mv110_in_4_shasn_reserve_input, style: Lamp-Lamp1-Red
    Line (54,254) (199,254), colour toggle: PLC_PRG.mv110_in_6_shasn_left
    Line (301,255) (767,255), colour toggle: PLC_PRG.mv110_in_5_shasn_right
    Line (460,155) (460,190), invisible if: NOT(PLC_PRG.mv110_in_8_shasn_main)
    Line (460,189) (435,155), invisible if: PLC_PRG.mv110_in_8_shasn_main
    Line (588,155) (588,190), invisible if: NOT(PLC_PRG.mv110_in_9_shasn_reserve)
    Line (587,190) (612,155), invisible if: PLC_PRG.mv110_in_9_shasn_reserve
    hotkey  Id=481037385728, Key=KeyDown=True, KeyName=0, VisuElemId=5
    hotkey  Id=481038434304, Key=KeyName=0, VisuElemId=5
END_VISUALIZATION

// Device/Application/ips_1
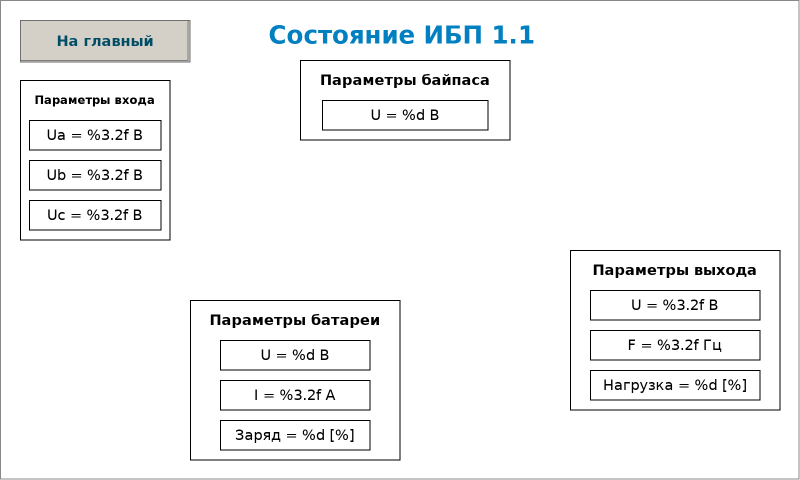
VISUALIZATION ips_1  // 800x480, background image ImagePool.ips_state_bg
    Rectangle (250,20 304x30), "Состояние ИБП 1.1"
    Button (20,20 170x42), "На главный"
        OnMouseClick:  Assign=main, Type=Assignment
    Rectangle (220,340 150x30), "U = %d В", text variable: PLC_PRG.ips1_battery_v
    Rectangle (220,380 150x30), "I = %3.2f A", text variable: PLC_PRG.ips1_battery_i_real
    Rectangle (220,420 150x30), "Заряд = %d [%]", text variable: PLC_PRG.ips1_battery_capacity
    Rectangle (590,290 170x30), "U = %3.2f В", text variable: PLC_PRG.ips1_out_v_real
    Rectangle (590,370 170x30), "Нагрузка = %d [%]", text variable: PLC_PRG.ips1_out_load_real
    Rectangle (570,250 210x160)
    Rectangle (580,260 190x20), "Параметры выхода"
    Rectangle (590,330 170x30), "F = %3.2f Гц", text variable: PLC_PRG.ips1_out_freq_real
    Rectangle (322,100 166x30), "U = %d В", text variable: PLC_PRG.ips1_bypass_v_real
    Rectangle (300,60 210x80)
    Rectangle (305,70 200x20), "Параметры байпаса"
    Rectangle (29,120 132x30), "Ua = %3.2f В", text variable: PLC_PRG.ips1_in_v_1_real
    Rectangle (29,160 132x30), "Ub = %3.2f В", text variable: PLC_PRG.ips1_in_v_2_real
    Rectangle (29,200 132x30), "Uc = %3.2f В", text variable: PLC_PRG.ips1_in_v_3_real
    Rectangle (20,80 150x160)
    Rectangle (25,90 140x20), "Параметры входа"
    Rectangle (190,300 210x160)
    Rectangle (195,310 200x20), "Параметры батареи"
    hotkey  Id=481037385728, Key=KeyDown=True, KeyName=0, VisuElemId=3
    hotkey  Id=481038434304, Key=KeyName=0, VisuElemId=3
END_VISUALIZATION

// Device/Application/ips_2
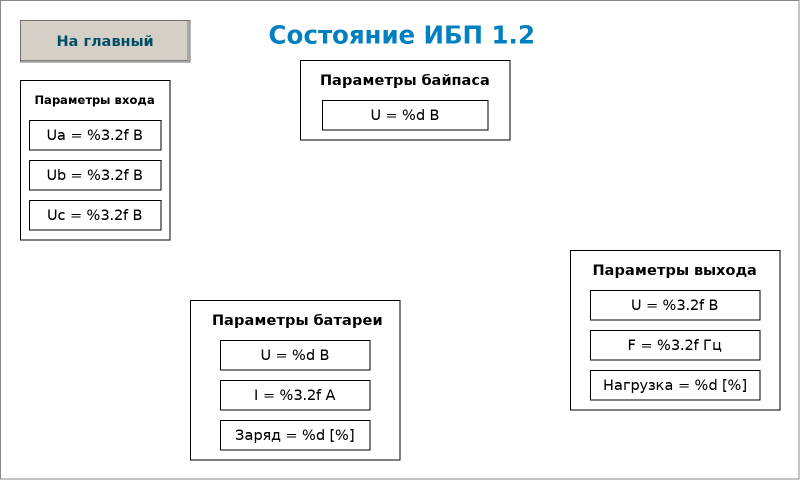
VISUALIZATION ips_2  // 800x480, background image ImagePool.ips_state_bg
    Rectangle (250,20 304x30), "Состояние ИБП 1.2"
    Button (20,20 170x42), "На главный"
        OnMouseClick:  Assign=main, Type=Assignment
    Rectangle (220,340 150x30), "U = %d В", text variable: PLC_PRG.ips2_battery_v
    Rectangle (220,380 150x30), "I = %3.2f A", text variable: PLC_PRG.ips2_battery_i_real
    Rectangle (220,420 150x30), "Заряд = %d [%]", text variable: PLC_PRG.ips2_battery_capacity
    Rectangle (590,290 170x30), "U = %3.2f В", text variable: PLC_PRG.ips2_out_v_real
    Rectangle (590,370 170x30), "Нагрузка = %d [%]", text variable: PLC_PRG.ips2_out_load_real
    Rectangle (570,250 210x160)
    Rectangle (580,260 190x20), "Параметры выхода"
    Rectangle (590,330 170x30), "F = %3.2f Гц", text variable: PLC_PRG.ips2_out_freq_real
    Rectangle (322,100 166x30), "U = %d В", text variable: PLC_PRG.ips2_bypass_v_real
    Rectangle (300,60 210x80)
    Rectangle (310,70 190x20), "Параметры байпаса"
    Rectangle (29,120 132x30), "Ua = %3.2f В", text variable: PLC_PRG.ips2_in_v_1_real
    Rectangle (29,160 132x30), "Ub = %3.2f В", text variable: PLC_PRG.ips2_in_v_2_real
    Rectangle (29,200 132x30), "Uc = %3.2f В", text variable: PLC_PRG.ips2_in_v_3_real
    Rectangle (20,80 150x160)
    Rectangle (25,90 140x20), "Параметры входа"
    Rectangle (190,300 210x160)
    Rectangle (205,310 185x20), "Параметры батареи"
    hotkey  Id=481037385728, Key=KeyDown=True, KeyName=0, VisuElemId=3
    hotkey  Id=481038434304, Key=KeyName=0, VisuElemId=3
END_VISUALIZATION

// Device/Application/alarms
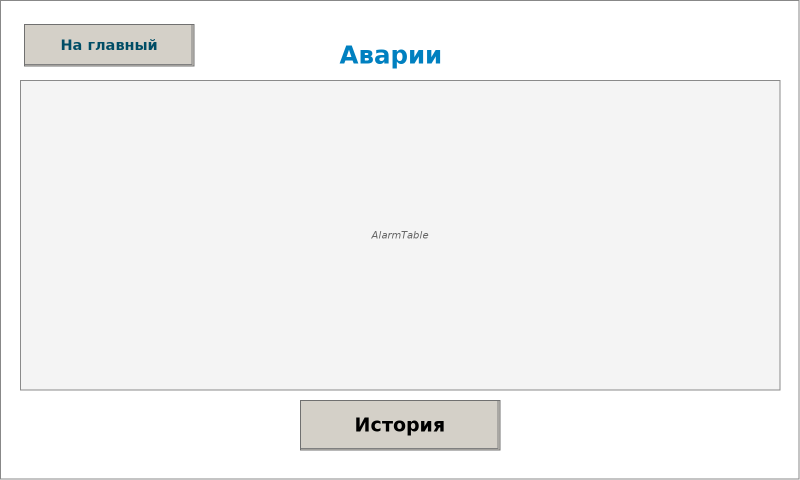
VISUALIZATION alarms  // 800x480, background image ImagePool.bg_800
    Rectangle (230,40 322x30), "Аварии"
    Button (24,24 170x42), "На главный"
        OnMouseClick:  Assign=main, Type=Assignment
    AlarmTable (20,80 760x310)
        Column[0]: ColumnTitle=Время
        Column[1]: ColumnTitle=Сообщение
        p1521930926: __All
        p1663851261: __All
        p428520879: PLC_PRG.ack
        p3266827225: PLC_PRG.history
    Button (300,400 200x50), "История", colour toggle: PLC_PRG.history
        toggle PLC_PRG.history
    hotkey  Id=481037385728, Key=KeyDown=True, KeyName=0, VisuElemId=3
    hotkey  Id=481038434304, Key=KeyName=0, VisuElemId=3
END_VISUALIZATION

// Device/Application/log_data
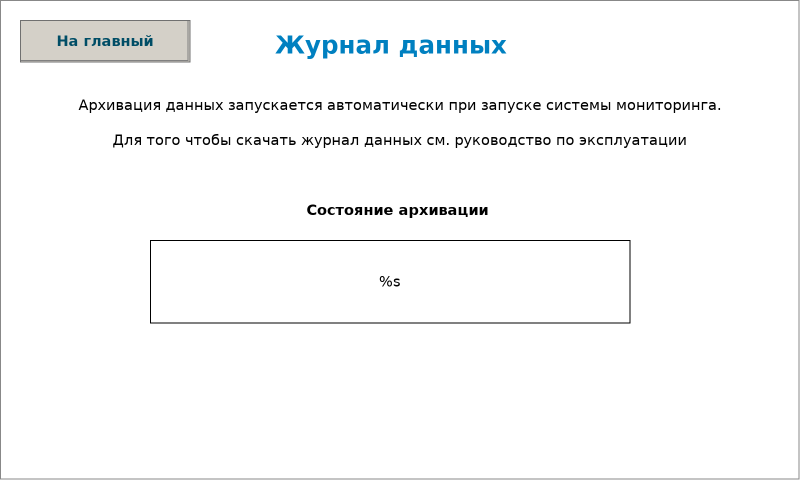
VISUALIZATION log_data  // 800x480, background image ImagePool.bg_800
    Rectangle (230,30 322x30), "Журнал данных"
    Button (20,20 170x42), "На главный"
        OnMouseClick:  Assign=main, Type=Assignment
    Rectangle (150,240 480x83), "%s", text variable: LogSaver.INFO
    Label (25,90 750x30), "Архивация данных запускается автоматически при запуске системы мониторинга."
    Label (25,125 750x30), "Для того чтобы скачать журнал данных см. руководство по эксплуатации"
    Label (210,195 375x30), "Состояние архивации"
    hotkey  Id=481037385728, Key=KeyDown=True, KeyName=0, VisuElemId=3
    hotkey  Id=481038434304, Key=KeyName=0, VisuElemId=3
END_VISUALIZATION

// Device/Application/SHOPS
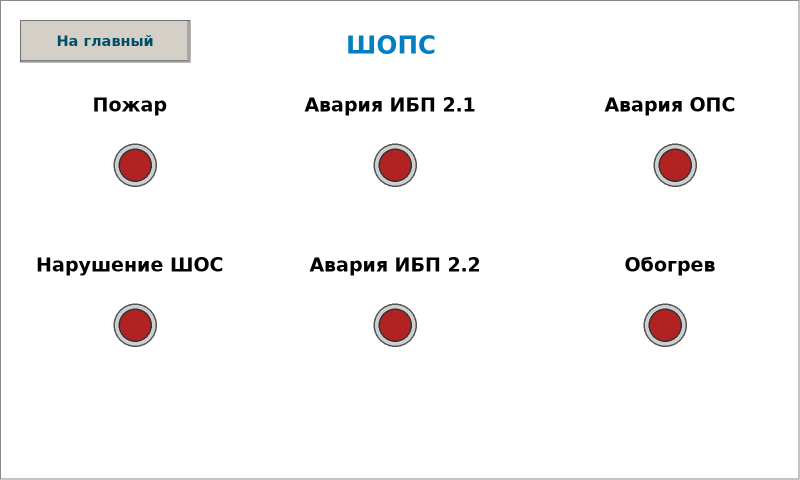
VISUALIZATION SHOPS  // 800x480, background image ImagePool.bg_800
    Rectangle (230,30 322x30), "ШОПС"
    Button (20,20 170x42), "На главный"
        OnMouseClick:  Assign=main, Type=Assignment
    Lamp1 (110,140 50x50), variable: PLC_PRG.mv110_in_1_fire, style: Lamp-Lamp1-Red
    Rectangle (20,90 220x30), "Пожар"
    Lamp1 (110,300 50x50), variable: PLC_PRG.mv110_in_0_alarm_shos, style: Lamp-Lamp1-Red
    Rectangle (20,250 220x30), "Нарушение ШОС"
    Lamp1 (650,140 50x50), variable: PLC_PRG.mv110_in_2_alarm_ops, style: Lamp-Lamp1-Red
    Rectangle (560,90 220x30), "Авария ОПС"
    Lamp1 (370,140 50x50), variable: PLC_PRG.mpx1_alarm, style: Lamp-Lamp1-Red
    Rectangle (280,90 220x30), "Авария ИБП 2.1"
    Lamp1 (370,300 50x50), variable: PLC_PRG.mpx2_alarm, style: Lamp-Lamp1-Red
    Rectangle (280,250 230x30), "Авария ИБП 2.2"
    Lamp1 (640,300 50x50), variable: PLC_PRG.mv110_in_7_heating, style: Lamp-Lamp1-Red
    Rectangle (560,250 220x30), "Обогрев"
    hotkey  Id=481037385728, Key=KeyDown=True, KeyName=0, VisuElemId=3
    hotkey  Id=481038434304, Key=KeyName=0, VisuElemId=3
END_VISUALIZATION

(* text list AlarmGroup (id | default)
  44 | Отсутствует напряжение на секции
  43 | Отсутствует напряжение на вводе №2
  42 | Отсутствует напряжение на вводе №1
  41 | Пониженное напряжение  на секции №2 Uc = TRIGGERVALUE
  40 | Повышенное напряжение  на секции №2 Uc = TRIGGERVALUE
  39 | Пониженное напряжение на секции №2 Ub = TRIGGERVALUE
  38 | Повышенное напряжение  на секции №2 Ub = TRIGGERVALUE
  37 | Пониженное напряжение на секции №2 Ua = TRIGGERVALUE
  36 | Повышенное напряжение на секции №2 Ua = TRIGGERVALUE
  35 | Пониженное напряжение на секции №1 Uc = TRIGGERVALUE
  34 | Повышенное напряжение на секции №1 Uc = TRIGGERVALUE
  33 | Пониженное напряжение на секции №1 Ub = TRIGGERVALUE
  32 | Повышенное напряжение на секции №1 Ub = TRIGGERVALUE
  31 | Пониженное напряжени на секции №1 Ua = TRIGGERVALUE
  30 | Повышенное напряжение на секции №1 Ua = TRIGGERVALUE
  29 | Перегрузка Ic на секции шин
  28 | Перегрузка Ib на секции шин
  27 | Перегрузка Ia  на секции шин
  26 | Перегрузка Ic на вводе №2
  25 | Перегрузка Ib на вводе №2
  24 | Перегрузка Ia на вводе №2
  23 | Пониженное напряжение на вводе №2 Uc = TRIGGERVALUE
  22 | Повышенное напряжение на вводе №2 Uc = TRIGGERVALUE
  21 | Пониженное напряжение на вводе №2 Ub = TRIGGERVALUE
  20 | Превышена максимальная температура
  19 | Нет связи с ЩРПА, ШАСН, ШОПС
  18 | Нет связи с ИБПС 2.2
  17 | Нет связи с ИБПС 2.1
  16 | Нет связи с ИБПА 1.2
  15 | Нет связи с ИБПА 1.1
  14 | Обогрев
  13 | Авария ИБПC 2.2
  12 | Авария ИБПC 2.1
  11 | Авария ОПС
  10 | Нарушение ШОС
  9 | Пожар
  8 | Авария ввода №2
  7 | Авария ввода №1
  6 | Авария секционного автомата
  5 | Пониженное напряжение
  4 | Ошибка_2
  3 | Ошибка_1
  2 | Предупреждение_3
  1 | Предупреждение_2
  0 | Предупреждение_1
   |  *)
